(* PLC project LMM.project, Inovance company InoProShop(V1.9.1.6) InoProShop(V1.9.1.6) *)
(* stored: creationDateTime 2026-08-05T19:09:37.7446622, modificationDateTime 2026-08-05T19:09:08.6866302 *)

VAR_GLOBAL  (* GVL *)
  StartBtn AT %IX1.6 : BOOL;  (* 【面板启动】→ HMI_xStart *)
  StopBtn AT %IX1.4 : BOOL;  (* 【面板停止】→ HMI_xStop *)
  ResetBtn : BOOL;  (* 【面板复位】→ HMI_xStopHold3s；地址现场另绑 *)
  EStop AT %IX0.4 : BOOL;  (* 【面板急停】正常=TRUE 按下=FALSE *)
  StopLamp AT %QX0.6 : BOOL;  (* 【停止指示灯】← Dev_xStop *)
  StartLamp AT %QX0.7 : BOOL;  (* 【运行指示灯】← Dev_xRun *)
  JogFwd : BOOL;  (* 【面板前进】手动 X+ *)
  JogBwd : BOOL;  (* 【面板后退】手动 X- *)
  JogRight : BOOL;  (* 【面板右】手动 Y+ *)
  JogLeft : BOOL;  (* 【面板左】手动 Y- *)
  JogUp : BOOL;  (* 【面板上】手动 Z+ *)
  JogDown : BOOL;  (* 【面板下】手动 Z- *)
  JogClockAdd : BOOL;  (* 【面板顺时针】手动 R+ *)
  JogClockMis : BOOL;  (* 【面板逆时针】手动 R- *)
  HMI_xEStop : BOOL;  (* 【急停】TRUE正常 FALSE按下 = 物理 AND 触摸屏Req AND Web *)
  HMI_xStop : BOOL;  (* 【停止】任一源为真即停；长按3s=复位 *)
  HMI_xStopHold3s : BOOL;  (* 【复位】清急停锁存 + 轴故障复位 *)
  HMI_xStart : BOOL;  (* 【启动】上升沿 *)
  HMI_xEnable : BOOL;  (* 【启动别名】与 HMI_xStart 等效 *)
  xEStopLatched : BOOL;  (* 【急停锁存】仅复位可清 *)
  xFaultAggregate : BOOL;  (* 【故障汇总】任轴 ErrorStop *)
  eCtrlSrc : INT;  (* 【控制源】0=面板/触摸屏 1=远程Web；仅 PRG_TcpHmi 写 *)
  eOpMode : INT;  (* 【运行方式】0手动 1自动 *)
  iAlarmID : INT;  (* 【内部报警号】 *)
  HMI_eDevState : INT;  (* 【只读·状态码】0停 1运行 2错误 *)
  HMI_eOpMode : INT;  (* 【只读·方式显示】0手动 1自动 *)
  HMI_iAlarmShow : INT;  (* 【只读·报警号】1001急停 1002轴故障 1005力超时 1006从站失败 1007未就绪；1008已废 *)
  Dev_xStop : BOOL;  (* 【内部·停止派生】 *)
  Dev_xRun : BOOL;  (* 【内部·运行派生】 *)
  Dev_xError : BOOL;  (* 【内部·故障派生】 *)
  HMI_xDevStop : BOOL;  (* 【只读·停止灯】 *)
  HMI_xDevRun : BOOL;  (* 【只读·运行灯】 *)
  HMI_xDevError : BOOL;  (* 【只读·故障灯】 *)
  HMI_xLampEStop : BOOL;  (* 【只读·急停指示】 *)
  HMI_xLampEnableOk : BOOL;  (* 【只读·就绪灯】 *)
  HMI_xLampFault : BOOL;  (* 【只读·故障指示】 *)
  HMI_xAutoMode : BOOL;  (* 【模式】FALSE手动 TRUE自动 *)
  HMI_xJogXPos : BOOL;  (* 【X+】M1=M2 同速同向；与旋转互斥 *)
  HMI_xJogXNeg : BOOL;  (* 【X-】 *)
  HMI_xSpinLeft : BOOL;  (* 【左旋转】差速原地转；与 X± 互斥 *)
  HMI_xSpinRight : BOOL;  (* 【右旋转】 *)
  HMI_xJogYPos : BOOL;  (* 【Y+】受限位 *)
  HMI_xJogYNeg : BOOL;  (* 【Y-】 *)
  HMI_xJogZPos : BOOL;  (* 【Z+】回零后软限位 [-0.7,0] *)
  HMI_xJogZNeg : BOOL;  (* 【Z-】 *)
  HMI_xJogRPos : BOOL;  (* 【R+】需 xM5Ready *)
  HMI_xJogRNeg : BOOL;  (* 【R-】 *)
  HMI_xHomeY : BOOL;  (* 【Y回零】 *)
  HMI_xHomeZ : BOOL;  (* 【Z回零】完成后软限位生效 *)
  HMI_xHomeR : BOOL;  (* 【R回零】编码器回零 *)
  HMI_iHomeAxis : INT := 0;  (* 【回零轴选择】0无 1Y 2Z 3R *)
  HMI_xHomeExec : BOOL;  (* 【回零执行】对选定轴 *)
  HMI_xHomedY : BOOL;  (* 【只读·Y已回零】 *)
  HMI_xHomedZ : BOOL;  (* 【只读·Z已回零】 *)
  HMI_xHomedR : BOOL;  (* 【只读·R已回零】 *)
  HMI_xHomeBusyY : BOOL;  (* 【只读·Y回零中】 *)
  HMI_xHomeBusyZ : BOOL;  (* 【只读·Z回零中】 *)
  HMI_xHomeBusyR : BOOL;  (* 【只读·R回零中】 *)
  HMI_xAutoStart : BOOL;  (* 【自动启动】上升沿 *)
  HMI_xAutoAbort : BOOL;  (* 【自动中止】立即结束 *)
  HMI_rHeadingErr : REAL := 0.0;  (* 【航向误差】视觉/外部纠偏输入（实时量，不保持） *)
  iAutoStep : INT;  (* 【自动步】0Idle..6Done *)
  HMI_iAutoStepShow : INT;  (* 【只读·自动步号】 *)
  HMI_xAutoBusy : BOOL;  (* 【只读·自动忙】 *)
  HMI_xAutoDone : BOOL;  (* 【只读·自动完成】 *)
  Force_xEnable : BOOL := TRUE;  (* 【力通讯总使能】 *)
  Force_wInRaw AT %IW102 : WORD;  (* 组态读通道：0x0000 原始力 *)
  Force_wOutTare AT %QW42 : WORD;  (* 组态写通道：0x0011 去皮 *)
  Force_wOutUnit AT %QW43 : WORD := 5;  (* 组态写通道：0x0002 单位 5=N *)
  Force_rScale : REAL := 0.01;  (* 原始值倍率 *)
  Force_xReadTrig : BOOL;  (* 【内部·力读触发】组态用，勿绑屏 *)
  Force_xCommOk : BOOL;  (* 【只读·力通讯正常】 *)
  Force_xTimeout : BOOL;  (* 【只读·力超时】报警1005 *)
  Force_xSlaveFail : BOOL;  (* 【只读·从站使能失败】报警1006 *)
  Force_xTareBusy : BOOL;  (* 【只读·去皮中】 *)
  Force_xTareDone : BOOL;  (* 【只读·去皮完成】 *)
  Force_iRaw : INT;  (* 【只读·原始计数】 *)
  Force_iState : INT;  (* 【只读·力任务状态】 *)
  rForceAct : REAL;  (* 【实际力】N；Axis 任务写（模拟时 Logic 写） *)
  rForceKp : REAL;  (* 【内部·恒力Kp】 *)
  HMI_rForceSim : REAL;  (* 【力模拟值】N *)
  HMI_xForceSimEnable : BOOL;  (* 【力模拟使能】台架用 *)
  HMI_xForceTare : BOOL;  (* 【去皮】上升沿 *)
  HMI_xForceUntare : BOOL;  (* 【取消去皮】上升沿 *)
  HMI_xForceGuide : BOOL;  (* 【力引导电平】TRUE 持续 Z 恒力跟随 *)
  HMI_rForceShow : REAL;  (* 【只读·显示力】N *)
  Logic_xForceTare : BOOL;  (* 【内部·自动步去皮脉冲】 *)
  I_xLimYPos : BOOL;  (* 【Y正限位开关】 *)
  I_xLimYNeg : BOOL;  (* 【Y负限位开关】 *)
  I_xLimZPos : BOOL;  (* 【Z正限位开关】 *)
  I_xLimZNeg : BOOL;  (* 【Z负限位开关】 *)
  xIlk_BlockYPlus : BOOL;  (* 【联锁禁Y+】开关 ∨ Cfg 限位 *)
  xIlk_BlockYNeg : BOOL;  (* 【联锁禁Y-】 *)
  xIlk_BlockZPlus : BOOL;  (* 【联锁禁Z+】 *)
  xIlk_BlockZNeg : BOOL;  (* 【联锁禁Z-】 *)
  xM5Ready : BOOL := TRUE;  (* 【第5轴就绪】FALSE=忽略 R *)
  AxisCmd_xPower : BOOL;  (* 【轴使能】= 安全条件 *)
  AxisCmd_xStopAll : BOOL;  (* 【全停】急停/停止/故障/中止 *)
  AxisCmd_xResetFault : BOOL;  (* 【故障复位脉冲】 *)
  AxisCmd_xJogXPos : BOOL;  (* 【X+】 *)
  AxisCmd_xJogXNeg : BOOL;  (* 【X-】 *)
  AxisCmd_xSpinLeft : BOOL;  (* 【左旋】 *)
  AxisCmd_xSpinRight : BOOL;  (* 【右旋】 *)
  AxisCmd_xJogYPos : BOOL;  (* 【Y+】 *)
  AxisCmd_xJogYNeg : BOOL;  (* 【Y-】 *)
  AxisCmd_xJogZPos : BOOL;  (* 【Z+】 *)
  AxisCmd_xJogZNeg : BOOL;  (* 【Z-】 *)
  AxisCmd_xJogRPos : BOOL;  (* 【R+】 *)
  AxisCmd_xJogRNeg : BOOL;  (* 【R-】 *)
  AxisCmd_xHomeY : BOOL;  (* 【Y回零】完成/停止清 *)
  AxisCmd_xHomeZ : BOOL;  (* 【Z回零】 *)
  AxisCmd_xHomeR : BOOL;  (* 【R回零】 *)
  AxisCmd_xMoveRelX : BOOL;  (* 【X相对走距】速度模式+里程判完成 *)
  AxisCmd_rMoveDistX : REAL;  (* 【X相对距离】 *)
  AxisCmd_rMoveVelX : REAL;  (* 【X相对速度】 *)
  AxisCmd_xMoveRelY : BOOL;  (* 【Y相对】 *)
  AxisCmd_rMoveDistY : REAL;  (* 【Y相对距离】自动=跨距 *)
  AxisCmd_rMoveVelY : REAL;  (* 【Y速度】 *)
  AxisCmd_xMoveAbsY : BOOL;  (* 【Y绝对】归位用 *)
  AxisCmd_rMoveAbsPosY : REAL;  (* 【Y绝对目标】 *)
  AxisCmd_xForceFollow : BOOL;  (* 【Z力跟随】 *)
  AxisCmd_rForceSet : REAL;  (* 【力目标】 *)
  AxisCmd_rForceKp : REAL;  (* 【力Kp】 *)
  AxisCmd_rForceVelMax : REAL;  (* 【力跟随限速】 *)
  AxisCmd_xHoldR : BOOL;  (* 【R保持角】 *)
  AxisCmd_rRHoldPos : REAL;  (* 【R保持角位置】 *)
  AxisCmd_rHeadingErr : REAL;  (* 【航向误差】 *)
  AxisCmd_rTrackKp : REAL;  (* 【纠偏Kp】 *)
  AxisCmd_rJogVelX : REAL;  (* 【X点动速度】 *)
  AxisCmd_rSpinVel : REAL := 0.0;  (* 【旋转速度】 *)
  AxisCmd_rJogVelY : REAL;  (* 【Y点动速度】 *)
  AxisCmd_rJogVelZ : REAL;  (* 【Z点动速度】 *)
  AxisCmd_rJogVelR : REAL;  (* 【R点动速度】 *)
  AxisCmd_rWheelBase : REAL;  (* 【跨距】限幅 4..6 *)
  AxisCmd_rAccX : REAL;  (* 【X加速度】 *)
  AxisCmd_rDecX : REAL;  (* 【X减速度】 *)
  AxisCmd_rAccY : REAL;  (* 【Y加速度】 *)
  AxisCmd_rDecY : REAL;  (* 【Y减速度】 *)
  AxisCmd_rAccZ : REAL;  (* 【Z加速度】 *)
  AxisCmd_rDecZ : REAL;  (* 【Z减速度】 *)
  AxisCmd_rAccR : REAL;  (* 【R加速度】 *)
  AxisCmd_rDecR : REAL;  (* 【R减速度】 *)
  AxisFb_rVelCmdM1 : REAL;  (* 【只读·M1速度指令】含纠偏/旋转 *)
  AxisFb_rVelCmdM2 : REAL;  (* 【只读·M2速度指令】 *)
  AxisFb_rPosM1 : REAL;  (* 【只读·M1位置】 *)
  AxisFb_rPosM2 : REAL;  (* 【只读·M2位置】 *)
  AxisFb_rPosX : REAL;  (* 【只读·Virtual X 位置】走距判据 *)
  AxisFb_rSyncErr : REAL;  (* 【只读·M1-M2 同步误差】 *)
  AxisFb_rVelFactorX : REAL;  (* 【只读·Virtual Override 倍率】 *)
  AxisFb_xGantryCoupled : BOOL;  (* 【只读·龙门已 GearIn】M1且M2 *)
  AxisFb_xInGearM1 : BOOL;  (* 【只读·M1 电子齿轮 InGear】 *)
  AxisFb_xInGearM2 : BOOL;  (* 【只读·M2 电子齿轮 InGear】 *)
  AxisFb_xPoweredV : BOOL;  (* 【只读·Virtual 已使能】 *)
  AxisFb_xSyncWarn : BOOL;  (* 【只读·同步预警】 *)
  AxisFb_xSyncFault : BOOL;  (* 【只读·同步跳闸】已废，恒 FALSE *)
  AxisFb_iGantryState : INT;  (* 【只读·0Idle 1Coupling 2Coupled 3Decouple 4Diff 5Align】 *)
  AxisFb_rPosY : REAL;  (* 【只读·Y位置】 *)
  AxisFb_rPosZ : REAL;  (* 【只读·Z位置】 *)
  AxisFb_rPosR : REAL;  (* 【只读·R位置/角度】 *)
  AxisFb_xStandstill1 : BOOL;  (* 【只读·M1静止】 *)
  AxisFb_xStandstill2 : BOOL;  (* 【只读·M2静止】 *)
  AxisFb_xStandstillY : BOOL;  (* 【只读·Y静止】 *)
  AxisFb_xStandstillZ : BOOL;  (* 【只读·Z静止】 *)
  AxisFb_xStandstillR : BOOL;  (* 【只读·R静止】 *)
  AxisFb_xMovingM1 : BOOL;  (* 【只读·M1运动中】 *)
  AxisFb_xMovingM2 : BOOL;  (* 【只读·M2运动中】 *)
  AxisFb_xMovingY : BOOL;  (* 【只读·Y运动中】 *)
  AxisFb_xMovingZ : BOOL;  (* 【只读·Z运动中】 *)
  AxisFb_xMovingR : BOOL;  (* 【只读·R运动中】 *)
  AxisFb_xPoweredM1 : BOOL;  (* 【只读·M1已使能】 *)
  AxisFb_xPoweredM2 : BOOL;  (* 【只读·M2已使能】 *)
  AxisFb_xPoweredY : BOOL;  (* 【只读·Y已使能】 *)
  AxisFb_xPoweredZ : BOOL;  (* 【只读·Z已使能】 *)
  AxisFb_xPoweredR : BOOL;  (* 【只读·R已使能】 *)
  AxisFb_xReadyM1 : BOOL;  (* 【只读·M1就绪】 *)
  AxisFb_xReadyM2 : BOOL;  (* 【只读·M2就绪】 *)
  AxisFb_xReadyY : BOOL;  (* 【只读·Y就绪】 *)
  AxisFb_xReadyZ : BOOL;  (* 【只读·Z就绪】 *)
  AxisFb_xReadyR : BOOL;  (* 【只读·R就绪】 *)
  AxisFb_xReady : BOOL;  (* 【只读·全轴就绪】FALSE → 报警1007 *)
  AxisFb_xHomedY : BOOL;  (* 【只读·Y已回零】 *)
  AxisFb_xHomedZ : BOOL;  (* 【只读·Z已回零】 *)
  AxisFb_xHomedR : BOOL;  (* 【只读·R已回零】 *)
  AxisFb_xFaultM1 : BOOL;  (* 【只读·M1故障】 *)
  AxisFb_xFaultM2 : BOOL;  (* 【只读·M2故障】 *)
  AxisFb_xFaultY : BOOL;  (* 【只读·Y故障】 *)
  AxisFb_xFaultZ : BOOL;  (* 【只读·Z故障】 *)
  AxisFb_xFaultR : BOOL;  (* 【只读·R故障】 *)
  AxisFb_xMoveDoneX : BOOL;  (* 【只读·X走距完成】 *)
  AxisFb_xMoveDoneY : BOOL;  (* 【只读·Y完成】 *)
  MB_CmdIn AT %IW103 : ARRAY[0..63] OF WORD;  (* 【命令入】Holding 1000..1063 *)
  MB_StatusOut AT %QW44 : ARRAY[0..63] OF WORD;  (* 【状态出】Holding 1100..1163 *)
  Tcp_iCommStatus : INT;  (* 【只读·通讯诊断】0离线 1在线 2版本错 3序号错 4超时 *)
  Tcp_xConnected : BOOL;  (* 【只读·远程已连接】 *)
  Tcp_xTimeout : BOOL;  (* 【只读·远程超时】 *)
  Tcp_xOnline : BOOL;  (* 【只读·远程在线可用】 *)
  Tcp_wLastHb : WORD;  (* 【内部·上次心跳】 *)
  Tcp_wLastSeq : WORD;  (* 【内部·上次命令序号】 *)
  Tcp_wStatusSeq : WORD;  (* 【内部·状态序号】 *)
  Tcp_xEStop : BOOL := TRUE;  (* 【Web影子·急停】掉线强制 TRUE *)
  Tcp_xStop : BOOL;  (* 【Web影子·停止】 *)
  Tcp_xStopHold3s : BOOL;  (* 【Web影子·复位】 *)
  Tcp_xStart : BOOL;  (* 【Web影子·启动】 *)
  Tcp_xEnable : BOOL;  (* 【Web影子·启动别名】 *)
  Tcp_xAutoMode : BOOL;  (* 【Web影子·模式】 *)
  Tcp_xJogXPos : BOOL;  (* 【Web影子·X+】 *)
  Tcp_xJogXNeg : BOOL;  (* 【Web影子·X-】 *)
  Tcp_xSpinLeft : BOOL;  (* 【Web影子·左旋】 *)
  Tcp_xSpinRight : BOOL;  (* 【Web影子·右旋】 *)
  Tcp_xJogYPos : BOOL;  (* 【Web影子·Y+】 *)
  Tcp_xJogYNeg : BOOL;  (* 【Web影子·Y-】 *)
  Tcp_xJogZPos : BOOL;  (* 【Web影子·Z+】 *)
  Tcp_xJogZNeg : BOOL;  (* 【Web影子·Z-】 *)
  Tcp_xJogRPos : BOOL;  (* 【Web影子·R+】 *)
  Tcp_xJogRNeg : BOOL;  (* 【Web影子·R-】 *)
  Tcp_xHomeY : BOOL;  (* 【Web影子·Y回零】 *)
  Tcp_xHomeZ : BOOL;  (* 【Web影子·Z回零】 *)
  Tcp_xHomeR : BOOL;  (* 【Web影子·R回零】 *)
  Tcp_iHomeAxis : INT := 0;  (* 【Web影子·回零轴选择】 *)
  Tcp_xHomeExec : BOOL;  (* 【Web影子·回零执行】 *)
  Tcp_rJogVelX : REAL := 0.4;  (* 【Web影子·X速度】 *)
  Tcp_rSpinVel : REAL := 0.3;  (* 【Web影子·旋转速度】 *)
  Tcp_rJogVelY : REAL := 0.3;  (* 【Web影子·Y速度】 *)
  Tcp_rJogVelZ : REAL := 0.2;  (* 【Web影子·Z速度】 *)
  Tcp_rJogVelR : REAL := 0.2;  (* 【Web影子·R速度】 *)
  Tcp_xAutoStart : BOOL;  (* 【Web影子·自动启动】 *)
  Tcp_xAutoAbort : BOOL;  (* 【Web影子·自动中止】 *)
  Tcp_rAutoDistX : REAL := 1.0;  (* 【Web影子·自动X距】 *)
  Tcp_rAutoVelX : REAL := 0.4;  (* 【Web影子·自动X速】 *)
  Tcp_rAutoVelY : REAL := 0.3;  (* 【Web影子·自动Y速】 *)
  Tcp_rAutoVelZ : REAL := 0.15;  (* 【Web影子·自动Z速】 *)
  Tcp_rWheelBase : REAL := 5.0;  (* 【Web影子·跨距】 *)
  Tcp_rForceSet : REAL := 100.0;  (* 【Web影子·力设定】 *)
  Tcp_xForceSimEnable : BOOL := FALSE;  (* 【Web影子·力模拟使能】 *)
  Tcp_rForceSim : REAL;  (* 【Web影子·力模拟值】 *)
  Tcp_xForceTare : BOOL;  (* 【Web影子·去皮】 *)
  Tcp_xForceUntare : BOOL;  (* 【Web影子·取消去皮】 *)
  Tcp_xForceGuide : BOOL;  (* 【Web影子·力引导】 *)
  Tcp_iAutoPasses : INT := 1;  (* 【Web影子·自动道数】 *)
  Tcp_rHeadingErr : REAL := 0.0;  (* 【Web影子·航向误差】 *)
  Tcp_rKpTrack : REAL;  (* 【Web影子·纠偏Kp】 *)
  Tcp_rKpForce : REAL;  (* 【Web影子·力Kp】 *)
  Tcp_rAccX : REAL := 100.0;  (* 【Web影子·X加速度】 *)
  Tcp_rDecX : REAL := 100.0;  (* 【Web影子·X减速度】 *)
  Tcp_rAccY : REAL := 100.0;  (* 【Web影子·Y加速度】 *)
  Tcp_rDecY : REAL := 100.0;  (* 【Web影子·Y减速度】 *)
  Tcp_rAccZ : REAL := 100.0;  (* 【Web影子·Z加速度】 *)
  Tcp_rDecZ : REAL := 100.0;  (* 【Web影子·Z减速度】 *)
  Tcp_rAccR : REAL := 100.0;  (* 【Web影子·R加速度】 *)
  Tcp_rDecR : REAL := 100.0;  (* 【Web影子·R减速度】 *)
  HMI_xStartReq : BOOL;  (* 【触摸屏启动】 *)
  HMI_xStopReq : BOOL;  (* 【触摸屏停止】 *)
  HMI_xResetReq : BOOL;  (* 【触摸屏复位】 *)
  HMI_xEStopReq : BOOL := TRUE;  (* 【触摸屏急停】TRUE正常 *)
  HMI_xAutoStartReq : BOOL;  (* 【触摸屏自动启动】 *)
  HMI_xAutoAbortReq : BOOL;  (* 【触摸屏自动中止】 *)
  {attribute 'retain'}
  HMI_rJogVelX : REAL := 0.4;  (* 【X直行速度】与旋转速度分开 *)
  {attribute 'retain'}
  HMI_rSpinVel : REAL := 0.3;  (* 【左右旋速度】 *)
  {attribute 'retain'}
  HMI_rJogVelY : REAL := 0.4;  (* 【Y点动速度】 *)
  {attribute 'retain'}
  HMI_rJogVelZ : REAL := 0.4;  (* 【Z点动速度】力跟随限速后备 *)
  {attribute 'retain'}
  HMI_rJogVelR : REAL := 0.2;  (* 【R点动速度】 *)
  {attribute 'retain'}
  HMI_rAccX : REAL := 25;  (* 【X加速度】 *)
  {attribute 'retain'}
  HMI_rDecX : REAL := 25;  (* 【X减速度】 *)
  {attribute 'retain'}
  HMI_rAccY : REAL := 25;  (* 【Y加速度】 *)
  {attribute 'retain'}
  HMI_rDecY : REAL := 25;  (* 【Y减速度】 *)
  {attribute 'retain'}
  HMI_rAccZ : REAL := 25;  (* 【Z加速度】 *)
  {attribute 'retain'}
  HMI_rDecZ : REAL := 25;  (* 【Z减速度】 *)
  {attribute 'retain'}
  HMI_rAccR : REAL := 25;  (* 【R加速度】 *)
  {attribute 'retain'}
  HMI_rDecR : REAL := 25;  (* 【R减速度】 *)
  {attribute 'retain'}
  HMI_rAutoDistX : REAL := 1.0;  (* 【自动X走距】每道 *)
  {attribute 'retain'}
  HMI_rAutoVelX : REAL := 0.4;  (* 【自动X速度】 *)
  {attribute 'retain'}
  HMI_rAutoVelY : REAL := 0.3;  (* 【自动Y速度】 *)
  {attribute 'retain'}
  HMI_rAutoVelZ : REAL := 0.15;  (* 【自动Z速度】力跟随限速参考 *)
  {attribute 'retain'}
  HMI_rWheelBase : REAL := 5.0;  (* 【龙门跨距=Y行程】4~6 m *)
  {attribute 'retain'}
  HMI_iAutoPasses : INT := 1;  (* 【自动总道数】≥1 *)
  {attribute 'retain'}
  HMI_rForceSet : REAL := 100.0;  (* 【恒力设定】N *)
  {attribute 'retain'}
  HMI_rKpForce : REAL := 1.0;  (* 【力跟随Kp】 *)
  {attribute 'retain'}
  HMI_rKpTrack : REAL := 0.0;  (* 【直线纠偏Kp】 *)
  {attribute 'retain'}
  Cfg_rLimYPos : REAL := 6.0;  (* 【Y正限位】m，默认跨距上限 *)
  {attribute 'retain'}
  Cfg_rLimYNeg : REAL := 0.0;  (* 【Y负限位】m *)
  {attribute 'retain'}
  Cfg_rLimZPos : REAL := 0.0;  (* 【Z正限位】上 *)
  {attribute 'retain'}
  Cfg_rLimZNeg : REAL := -0.7;  (* 【Z负限位】下压行程 *)
  {attribute 'retain'}
  Cfg_rLimRPos : REAL := 180.0;  (* 【R正限位】度 *)
  {attribute 'retain'}
  Cfg_rLimRNeg : REAL := -180.0;  (* 【R负限位】度 *)
  {attribute 'retain'}
  Cfg_rVelBaseMaxX : REAL := 1.0;  (* 【X速度基准】诊断倍率分母；≥最大 Jog/Auto *)
  {attribute 'retain'}
  Cfg_rPhaseMax : REAL := 0.01;  (* 【跟轨相位限幅】u；连续 Phasing *)
  {attribute 'retain'}
  Cfg_rSyncWarn : REAL := 0.02;  (* 【同步预警】|M1-M2|；降速 *)
  {attribute 'retain'}
  Cfg_rSyncFault : REAL := 0.05;  (* 【同步跳闸】已废；保留 RETAIN 布局 *)
END_VAR

PROGRAM PRG_Logic
  VAR
    tonHold : TON;
    tonReady : TON;
    xResetPulse : BOOL;
    xResetPrev : BOOL;
    xSafe : BOOL;
    xAutoStartPrev : BOOL;
    xAutoStartEdge : BOOL;
    rRHold : REAL;
    iPass : INT;
    xAutoTareSent : BOOL;
    xHomeTrigY : BOOL;
    xHomeTrigZ : BOOL;
    xHomeTrigR : BOOL;
    xHomeTrigYPrev : BOOL;
    xHomeTrigZPrev : BOOL;
    xHomeTrigRPrev : BOOL;
    xAnyHomeBusy : BOOL;
    xReadyAll : BOOL;
    xPanelSrc : BOOL;  (* eCtrlSrc=0：面板/触摸屏源 *)
    xJogXPosM : BOOL;  (* 合并后点动（HMI/Web OR 面板键） *)
    xJogXNegM : BOOL;
    xJogYPosM : BOOL;
    xJogYNegM : BOOL;
    xJogZPosM : BOOL;
    xJogZNegM : BOOL;
    xJogRPosM : BOOL;
    xJogRNegM : BOOL;
  END_VAR

            (* PRG_Logic — 消费已仲裁 HMI_* + 面板键；写 AxisCmd_*；状态只读派生（无状态机耦合）。
   禁止 CALL Axis / FB_Servo。 *)

(* ===== 急停锁存 / 长按复位 ===== *)
IF NOT HMI_xEStop THEN
    xEStopLatched := TRUE;
END_IF;
tonHold(IN := HMI_xStop AND HMI_xEStop, PT := T#3S);
xResetPulse := (HMI_xStopHold3s OR tonHold.Q) AND NOT xResetPrev;
xResetPrev := HMI_xStopHold3s OR tonHold.Q;
IF xResetPulse THEN
    xEStopLatched := FALSE;
    AxisCmd_xResetFault := TRUE;
    iAutoStep := 0;
    iPass := 0;
    Force_xSlaveFail := FALSE;
ELSE
    AxisCmd_xResetFault := FALSE;
END_IF;

(* 故障汇总：各轴 Errorstop（同步跳闸已废，不再 OR AxisFb_xSyncFault） *)
xFaultAggregate := AxisFb_xFaultM1 OR AxisFb_xFaultM2 OR AxisFb_xFaultY OR AxisFb_xFaultZ
    OR (xM5Ready AND AxisFb_xFaultR);

IF HMI_xAutoMode THEN eOpMode := 1; ELSE eOpMode := 0; END_IF;
HMI_eOpMode := eOpMode;

(* 安全 / 使能 —— 去耦：只看急停 + 故障 *)
xSafe := HMI_xEStop AND NOT xEStopLatched;
AxisCmd_xPower := xSafe;
AxisCmd_xStopAll := HMI_xStop OR NOT xSafe OR xFaultAggregate OR HMI_xAutoAbort;

(* 力/纠偏参数下发 *)
rForceKp := HMI_rKpForce;
IF rForceKp < 1.0E-6 THEN rForceKp := 1.0; END_IF;
AxisCmd_rForceSet := HMI_rForceSet;
AxisCmd_rForceKp := rForceKp;
AxisCmd_rForceVelMax := ABS(HMI_rAutoVelZ);
IF AxisCmd_rForceVelMax < 1.0E-6 THEN AxisCmd_rForceVelMax := ABS(HMI_rJogVelZ); END_IF;
AxisCmd_rHeadingErr := HMI_rHeadingErr;

IF HMI_xForceSimEnable THEN
    rForceAct := HMI_rForceSim;
END_IF;
HMI_rForceShow := rForceAct;

AxisCmd_rJogVelX := HMI_rJogVelX;
AxisCmd_rSpinVel := HMI_rSpinVel;
AxisCmd_rJogVelY := HMI_rJogVelY;
AxisCmd_rJogVelZ := HMI_rJogVelZ;
AxisCmd_rJogVelR := HMI_rJogVelR;
AxisCmd_rWheelBase := LIMIT(4.0, HMI_rWheelBase, 6.0);
(* 每轴加减速（RETAIN 参数；<1 时兜底 100） *)
AxisCmd_rAccX := HMI_rAccX; IF AxisCmd_rAccX < 1.0 THEN AxisCmd_rAccX := 100.0; END_IF;
AxisCmd_rDecX := HMI_rDecX; IF AxisCmd_rDecX < 1.0 THEN AxisCmd_rDecX := 100.0; END_IF;
AxisCmd_rAccY := HMI_rAccY; IF AxisCmd_rAccY < 1.0 THEN AxisCmd_rAccY := 100.0; END_IF;
AxisCmd_rDecY := HMI_rDecY; IF AxisCmd_rDecY < 1.0 THEN AxisCmd_rDecY := 100.0; END_IF;
AxisCmd_rAccZ := HMI_rAccZ; IF AxisCmd_rAccZ < 1.0 THEN AxisCmd_rAccZ := 100.0; END_IF;
AxisCmd_rDecZ := HMI_rDecZ; IF AxisCmd_rDecZ < 1.0 THEN AxisCmd_rDecZ := 100.0; END_IF;
AxisCmd_rAccR := HMI_rAccR; IF AxisCmd_rAccR < 1.0 THEN AxisCmd_rAccR := 100.0; END_IF;
AxisCmd_rDecR := HMI_rDecR; IF AxisCmd_rDecR < 1.0 THEN AxisCmd_rDecR := 100.0; END_IF;

(* 限位联锁：物理限位输入 ∨ 可配置硬限位（Cfg_rLim*，FB_Servo 内另有最终闸门） *)
xIlk_BlockYPlus := I_xLimYPos OR (AxisFb_rPosY >= Cfg_rLimYPos);
xIlk_BlockYNeg := I_xLimYNeg OR (AxisFb_rPosY <= Cfg_rLimYNeg);
xIlk_BlockZPlus := I_xLimZPos OR (AxisFb_rPosZ >= Cfg_rLimZPos);
xIlk_BlockZNeg := I_xLimZNeg OR (AxisFb_rPosZ <= Cfg_rLimZNeg);

(* 每拍清命令 *)
AxisCmd_xJogXPos := FALSE; AxisCmd_xJogXNeg := FALSE;
AxisCmd_xSpinLeft := FALSE; AxisCmd_xSpinRight := FALSE;
AxisCmd_xJogYPos := FALSE; AxisCmd_xJogYNeg := FALSE;
AxisCmd_xJogZPos := FALSE; AxisCmd_xJogZNeg := FALSE;
AxisCmd_xJogRPos := FALSE; AxisCmd_xJogRNeg := FALSE;
AxisCmd_xForceFollow := FALSE;
AxisCmd_xMoveRelX := FALSE;
AxisCmd_xMoveRelY := FALSE;
AxisCmd_xMoveAbsY := FALSE;
AxisCmd_xHoldR := FALSE;
AxisCmd_rTrackKp := 0.0;
Logic_xForceTare := FALSE;

xAutoStartEdge := HMI_xAutoStart AND NOT xAutoStartPrev;
xAutoStartPrev := HMI_xAutoStart;

IF HMI_xAutoAbort OR NOT xSafe OR xFaultAggregate THEN
    iAutoStep := 0;
    iPass := 0;
    HMI_xAutoBusy := FALSE;
END_IF;

(* ===== 点动源合并：面板键（仅面板/触摸屏源时）OR 触摸屏/Web ===== *)
xPanelSrc := (eCtrlSrc = 0);
xJogXPosM := HMI_xJogXPos OR (xPanelSrc AND JogFwd);
xJogXNegM := HMI_xJogXNeg OR (xPanelSrc AND JogBwd);
xJogYPosM := HMI_xJogYPos OR (xPanelSrc AND JogRight);
xJogYNegM := HMI_xJogYNeg OR (xPanelSrc AND JogLeft);
xJogZPosM := HMI_xJogZPos OR (xPanelSrc AND JogUp);
xJogZNegM := HMI_xJogZNeg OR (xPanelSrc AND JogDown);
xJogRPosM := HMI_xJogRPos OR (xPanelSrc AND JogClockAdd);
xJogRNegM := HMI_xJogRNeg OR (xPanelSrc AND JogClockMis);

(* ===== 手动 ===== *)
IF xSafe AND (eOpMode = 0) AND NOT HMI_xStop AND NOT xFaultAggregate THEN
    IF HMI_xSpinLeft XOR HMI_xSpinRight THEN
        AxisCmd_xSpinLeft := HMI_xSpinLeft;
        AxisCmd_xSpinRight := HMI_xSpinRight;
    ELSIF xJogXPosM XOR xJogXNegM THEN
        AxisCmd_xJogXPos := xJogXPosM;
        AxisCmd_xJogXNeg := xJogXNegM;
    END_IF;
    AxisCmd_xJogYPos := xJogYPosM AND NOT xIlk_BlockYPlus;
    AxisCmd_xJogYNeg := xJogYNegM AND NOT xIlk_BlockYNeg;
    IF HMI_xForceGuide THEN
        AxisCmd_xForceFollow := TRUE;
    ELSE
        AxisCmd_xJogZPos := xJogZPosM AND NOT xIlk_BlockZPlus;
        AxisCmd_xJogZNeg := xJogZNegM AND NOT xIlk_BlockZNeg;
    END_IF;
    IF xM5Ready THEN
        AxisCmd_xJogRPos := xJogRPosM;
        AxisCmd_xJogRNeg := xJogRNegM;
    END_IF;
END_IF;

(* ===== 自动多道循环 ===== *)
IF xSafe AND (eOpMode = 1) AND NOT HMI_xStop AND NOT xFaultAggregate THEN
    IF iAutoStep = 0 AND xAutoStartEdge THEN
        rRHold := AxisFb_rPosR;
        xAutoTareSent := FALSE;
        HMI_xAutoDone := FALSE;
        HMI_xAutoBusy := TRUE;
        iPass := 1;
        iAutoStep := 1;
    END_IF;

    CASE iAutoStep OF
        1:
            AxisCmd_xHoldR := TRUE;
            AxisCmd_rRHoldPos := rRHold;
            AxisCmd_rTrackKp := HMI_rKpTrack;
            AxisCmd_rMoveDistX := HMI_rAutoDistX;
            AxisCmd_rMoveVelX := HMI_rAutoVelX;
            AxisCmd_xMoveRelX := TRUE;
            IF AxisFb_xMoveDoneX THEN
                AxisCmd_xMoveRelX := FALSE;
                iAutoStep := 2;
            END_IF;
        2:
            AxisCmd_xHoldR := TRUE;
            AxisCmd_rRHoldPos := rRHold;
            AxisCmd_rMoveAbsPosY := 0.0;
            AxisCmd_rMoveVelY := HMI_rAutoVelY;
            AxisCmd_xMoveAbsY := TRUE;
            IF AxisFb_xStandstillY AND (ABS(AxisFb_rPosY) < 0.005) THEN
                AxisCmd_xMoveAbsY := FALSE;
                xAutoTareSent := FALSE;
                iAutoStep := 3;
            END_IF;
        3:
            AxisCmd_xHoldR := TRUE;
            AxisCmd_rRHoldPos := rRHold;
            IF NOT xAutoTareSent THEN
                Logic_xForceTare := TRUE;
                xAutoTareSent := TRUE;
            END_IF;
            AxisCmd_xForceFollow := TRUE;
            IF rForceAct >= HMI_rForceSet THEN
                iAutoStep := 4;
            END_IF;
        4:
            AxisCmd_xHoldR := TRUE;
            AxisCmd_rRHoldPos := rRHold;
            AxisCmd_xForceFollow := TRUE;
            AxisCmd_rMoveDistY := AxisCmd_rWheelBase;
            AxisCmd_rMoveVelY := HMI_rAutoVelY;
            AxisCmd_xMoveRelY := TRUE;
            IF AxisFb_xMoveDoneY THEN
                AxisCmd_xMoveRelY := FALSE;
                iAutoStep := 5;
            END_IF;
        5:
            IF iPass < HMI_iAutoPasses THEN
                iPass := iPass + 1;
                iAutoStep := 1;
            ELSE
                iAutoStep := 6;
            END_IF;
        6:
            HMI_xAutoBusy := FALSE;
            HMI_xAutoDone := TRUE;
            iAutoStep := 0;
            iPass := 0;
    END_CASE;
END_IF;

(* ===== 回零：Y/Z/R；同时只回一轴 ===== *)
xHomeTrigY := HMI_xHomeY OR ((HMI_iHomeAxis = 1) AND HMI_xHomeExec);
xHomeTrigZ := HMI_xHomeZ OR ((HMI_iHomeAxis = 2) AND HMI_xHomeExec);
xHomeTrigR := HMI_xHomeR OR ((HMI_iHomeAxis = 3) AND HMI_xHomeExec);
xAnyHomeBusy := AxisCmd_xHomeY OR AxisCmd_xHomeZ OR AxisCmd_xHomeR;

IF AxisCmd_xStopAll OR NOT xSafe OR xFaultAggregate THEN
    AxisCmd_xHomeY := FALSE;
    AxisCmd_xHomeZ := FALSE;
    AxisCmd_xHomeR := FALSE;
ELSE
    IF AxisCmd_xHomeY AND AxisFb_xHomedY THEN AxisCmd_xHomeY := FALSE; END_IF;
    IF AxisCmd_xHomeZ AND AxisFb_xHomedZ THEN AxisCmd_xHomeZ := FALSE; END_IF;
    IF AxisCmd_xHomeR AND AxisFb_xHomedR THEN AxisCmd_xHomeR := FALSE; END_IF;
    IF (eOpMode = 0) AND NOT HMI_xStop THEN
        IF xHomeTrigY AND NOT xHomeTrigYPrev AND NOT xAnyHomeBusy THEN
            AxisCmd_xHomeY := TRUE;
        ELSIF xHomeTrigZ AND NOT xHomeTrigZPrev AND NOT xAnyHomeBusy THEN
            AxisCmd_xHomeZ := TRUE;
        ELSIF xHomeTrigR AND NOT xHomeTrigRPrev AND NOT xAnyHomeBusy AND xM5Ready THEN
            AxisCmd_xHomeR := TRUE;
        END_IF;
    END_IF;
END_IF;
xHomeTrigYPrev := xHomeTrigY;
xHomeTrigZPrev := xHomeTrigZ;
xHomeTrigRPrev := xHomeTrigR;

IF AxisCmd_xHomeY THEN AxisCmd_xJogYPos := FALSE; AxisCmd_xJogYNeg := FALSE; END_IF;
IF AxisCmd_xHomeZ THEN AxisCmd_xJogZPos := FALSE; AxisCmd_xJogZNeg := FALSE; AxisCmd_xForceFollow := FALSE; END_IF;
IF AxisCmd_xHomeR THEN AxisCmd_xJogRPos := FALSE; AxisCmd_xJogRNeg := FALSE; END_IF;

HMI_xHomedY := AxisFb_xHomedY;
HMI_xHomedZ := AxisFb_xHomedZ;
HMI_xHomedR := AxisFb_xHomedR;
HMI_xHomeBusyY := AxisCmd_xHomeY;
HMI_xHomeBusyZ := AxisCmd_xHomeZ;
HMI_xHomeBusyR := AxisCmd_xHomeR;

(* 使能就绪诊断 → 1007 *)
xReadyAll := AxisFb_xReadyM1 AND AxisFb_xReadyM2 AND AxisFb_xReadyY AND AxisFb_xReadyZ
    AND (NOT xM5Ready OR AxisFb_xReadyR);
tonReady(IN := AxisCmd_xPower AND NOT xReadyAll AND NOT xFaultAggregate, PT := T#2S);

(* 报警 *)
IF xEStopLatched OR NOT HMI_xEStop THEN
    iAlarmID := 1001;
ELSIF AxisFb_xFaultM1 OR AxisFb_xFaultM2 OR AxisFb_xFaultY OR AxisFb_xFaultZ
        OR (xM5Ready AND AxisFb_xFaultR) THEN
    iAlarmID := 1002;
ELSIF tonReady.Q THEN
    iAlarmID := 1007;
ELSIF NOT HMI_xForceSimEnable AND Force_xSlaveFail THEN
    iAlarmID := 1006;
ELSIF NOT HMI_xForceSimEnable AND Force_xTimeout THEN
    iAlarmID := 1005;
ELSE
    iAlarmID := 0;
END_IF;

(* 状态灯（只读派生，不互锁） *)
Dev_xError := xFaultAggregate;
Dev_xRun := xSafe AND NOT HMI_xStop AND NOT xFaultAggregate;
Dev_xStop := NOT Dev_xRun AND NOT Dev_xError;
HMI_xDevError := Dev_xError;
HMI_xDevRun := Dev_xRun;
HMI_xDevStop := Dev_xStop;
IF Dev_xError THEN HMI_eDevState := 2;
ELSIF Dev_xRun THEN HMI_eDevState := 1;
ELSE HMI_eDevState := 0; END_IF;

HMI_iAutoStepShow := iAutoStep;
HMI_xLampEStop := xEStopLatched OR NOT HMI_xEStop;
HMI_xLampEnableOk := Dev_xRun;
HMI_xLampFault := xFaultAggregate;
HMI_iAlarmShow := iAlarmID;

StopLamp := Dev_xStop;
StartLamp := Dev_xRun;
          
END_PROGRAM

PROGRAM PRG_Force485
  VAR
    iSlaveStep : INT;
    iSlaveTry : INT;
    tonSlave : TON;
    wSnap : WORD;
    wRawLast : WORD;
    xTarePrev : BOOL;
    xUntarePrev : BOOL;
    xUnitInit : BOOL;
    diRaw : DINT;
    rTmp : REAL;
    xTareReq : BOOL;
  END_VAR

            (*==============================================================================
 * PRG_Force485 — SM1001 使能 + 发读等回文（最多3次）+ 去皮/换算
 *
 * 流程（严格按需求）：
 *   1) 使能 Modbus 从站 SM1001
 *   2) 发送一次读（破坏 Force_wInRaw 快照，等组态 FC03 通道写回 = 有回文）
 *   3) 有回文 → Force_xCommOk，进入成功态，不再重试
 *   4) 无回文 → 关闭 SM1001，重新使能，再读
 *   5) 3 次均无回文 → Force_xSlaveFail / 报警 1006
 *
 * 组态：读通道 FC03 0x0000 → Force_wInRaw（循环或由 Force_xReadTrig 触发均可）
 *============================================================================*)

Force_xTareDone := FALSE;

IF NOT Force_xEnable THEN
	SM1001 := FALSE;
	Force_xReadTrig := FALSE;
	Force_xCommOk := FALSE;
	Force_xTimeout := FALSE;
	Force_xTareBusy := FALSE;
	Force_xSlaveFail := FALSE;
	Force_iState := 0;
	iSlaveStep := 0;
	iSlaveTry := 0;
	RETURN;
END_IF;

CASE iSlaveStep OF
	0: (* 准备：先关从站，再进入使能 *)
		IF iSlaveTry >= 3 THEN
			SM1001 := FALSE;
			Force_xReadTrig := FALSE;
			Force_xSlaveFail := TRUE;
			Force_xTimeout := TRUE;
			Force_xCommOk := FALSE;
			Force_iState := -2;
			iSlaveStep := 99;
		ELSE
			SM1001 := FALSE;
			Force_xReadTrig := FALSE;
			Force_xCommOk := FALSE;
			tonSlave(IN := FALSE);
			tonSlave(IN := TRUE, PT := T#200MS);
			Force_iState := 0;
			iSlaveStep := 1;
		END_IF;

	1: (* 关断保持 *)
		SM1001 := FALSE;
		Force_xReadTrig := FALSE;
		tonSlave();
		IF tonSlave.Q THEN
			tonSlave(IN := FALSE);
			iSlaveStep := 2;
		END_IF;

	2: (* ① 使能从站 *)
		SM1001 := TRUE;
		Force_xReadTrig := FALSE;
		iSlaveTry := iSlaveTry + 1;
		tonSlave(IN := FALSE);
		tonSlave(IN := TRUE, PT := T#100MS);
		Force_iState := 1;
		iSlaveStep := 3;

	3: (* 使能稳定后：② 发读命令（破坏快照 + 读触发） *)
		SM1001 := TRUE;
		tonSlave();
		IF tonSlave.Q THEN
			(* 破坏映射值：有回文时通道会写回真实寄存器 *)
			wSnap := Force_wInRaw XOR 16#FFFF;
			Force_wInRaw := wSnap;
			Force_xReadTrig := FALSE;
			tonSlave(IN := FALSE);
			tonSlave(IN := TRUE, PT := T#20MS);
			Force_iState := 2;
			iSlaveStep := 4;
		END_IF;

	4: (* 读触发上升沿 *)
		SM1001 := TRUE;
		tonSlave();
		IF tonSlave.Q THEN
			Force_xReadTrig := TRUE;
			tonSlave(IN := FALSE);
			tonSlave(IN := TRUE, PT := T#500MS);
			Force_iState := 3;
			iSlaveStep := 5;
		END_IF;

	5: (* ③ 等回文：Force_wInRaw 被总线写回且不等于破坏值 *)
		SM1001 := TRUE;
		Force_xReadTrig := TRUE;
		tonSlave();
		IF Force_wInRaw <> wSnap THEN
			(* 有回文 → 成功，不再尝试 *)
			Force_xReadTrig := FALSE;
			Force_xCommOk := TRUE;
			Force_xTimeout := FALSE;
			Force_xSlaveFail := FALSE;
			wRawLast := Force_wInRaw;
			Force_iState := 4;
			tonSlave(IN := FALSE);
			iSlaveStep := 10;
		ELSIF tonSlave.Q THEN
			(* 无回文 → 关从站，回到 0 重新使能 *)
			Force_xReadTrig := FALSE;
			SM1001 := FALSE;
			Force_xCommOk := FALSE;
			Force_iState := 5;
			tonSlave(IN := FALSE);
			iSlaveStep := 0;
		END_IF;

	10: (* 成功：保持使能，不再重试使能 *)
		SM1001 := TRUE;
		Force_xReadTrig := FALSE;
		Force_xCommOk := TRUE;
		Force_xTimeout := FALSE;
		IF Force_wInRaw <> wRawLast THEN
			wRawLast := Force_wInRaw;
		END_IF;

	99: (* 3 次失败；复位清 Force_xSlaveFail 后从 0 重来 *)
		SM1001 := FALSE;
		Force_xReadTrig := FALSE;
		IF Force_xSlaveFail THEN
			Force_xTimeout := TRUE;
			Force_xCommOk := FALSE;
		ELSE
			iSlaveTry := 0;
			Force_xTimeout := FALSE;
			iSlaveStep := 0;
		END_IF;
END_CASE;

(* ----- 原始值换算（成功后持续；探测中也换算便于监视） ----- *)
diRaw := DWORD_TO_DINT(WORD_TO_DWORD(Force_wInRaw));
IF diRaw > 32767 THEN
	diRaw := diRaw - 65536;
END_IF;
Force_iRaw := DINT_TO_INT(diRaw);
IF Force_rScale < 1.0E-12 THEN
	rTmp := INT_TO_REAL(Force_iRaw);
ELSE
	rTmp := INT_TO_REAL(Force_iRaw) * Force_rScale;
END_IF;
IF NOT HMI_xForceSimEnable AND iSlaveStep = 10 THEN
	rForceAct := rTmp;
END_IF;

IF NOT xUnitInit AND iSlaveStep = 10 THEN
	Force_wOutUnit := 5;
	xUnitInit := TRUE;
END_IF;

xTareReq := FALSE;
IF iSlaveStep = 10 THEN
	IF ((HMI_xForceTare OR Tcp_xForceTare OR Logic_xForceTare) AND NOT xTarePrev) THEN
		Force_wOutTare := 1;
		xTareReq := TRUE;
		Force_xTareDone := TRUE;
	END_IF;
	xTarePrev := HMI_xForceTare OR Tcp_xForceTare OR Logic_xForceTare;
	IF Tcp_xForceTare THEN
		Tcp_xForceTare := FALSE;
	END_IF;
	IF Logic_xForceTare THEN
		Logic_xForceTare := FALSE;
	END_IF;

	IF ((HMI_xForceUntare OR Tcp_xForceUntare) AND NOT xUntarePrev) THEN
		Force_wOutTare := 2;
		xTareReq := TRUE;
		Force_xTareDone := TRUE;
	END_IF;
	xUntarePrev := HMI_xForceUntare OR Tcp_xForceUntare;
	IF Tcp_xForceUntare THEN
		Tcp_xForceUntare := FALSE;
	END_IF;
END_IF;

Force_xTareBusy := xTareReq;

          
END_PROGRAM

PROGRAM PLC_PRG

            (* MainTask 入口：HMI 交互 -> 设备逻辑；PRG_Axis_Control 在 ETHERCAT 任务独立运行 *)
PRG_TcpHmi();
PRG_Logic();
PRG_Force485();
          
END_PROGRAM

FUNCTION_BLOCK FB_XLineTrack
  VAR_INPUT
    xEnable : BOOL;
    xStop : BOOL;
    eMode : INT;
    rBaseVel : REAL;  (* 直行基础速度（可正可负） *)
    rSpinVel : REAL;  (* 原地旋转速度（正值） *)
    rHeadingErr : REAL;  (* 航向误差（视觉/外部；手动传 0） *)
    rKpTrack : REAL;  (* 纠偏 Kp *)
    rTrimMax : REAL;  (* 纠偏限幅 *)
  END_VAR
  VAR_OUTPUT
    rVelM1 : REAL;  (* M1 速度指令 *)
    rVelM2 : REAL;  (* M2 速度指令 *)
    xActive : BOOL;
  END_VAR
  VAR
    rTrim : REAL;
  END_VAR

            (* FB_XLineTrack — X 直行按航向误差纠偏差速 / 原地左右转。
   eMode: 0=无  1=直行(rBaseVel 带符号 + 纠偏)  2=左旋  3=右旋 *)

rTrim := LIMIT(-ABS(rTrimMax), rKpTrack * rHeadingErr, ABS(rTrimMax));

CASE eMode OF
    1:
        rVelM1 := rBaseVel + rTrim;
        rVelM2 := rBaseVel - rTrim;
    2:
        rVelM1 := ABS(rSpinVel);
        rVelM2 := -ABS(rSpinVel);
    3:
        rVelM1 := -ABS(rSpinVel);
        rVelM2 := ABS(rSpinVel);
ELSE
    rVelM1 := 0.0;
    rVelM2 := 0.0;
END_CASE;

IF xStop OR NOT xEnable THEN
    rVelM1 := 0.0;
    rVelM2 := 0.0;
END_IF;

xActive := (eMode <> 0) AND xEnable AND NOT xStop;
          
END_FUNCTION_BLOCK

FUNCTION_BLOCK FB_ForceFollow
  VAR_INPUT
    rForceSet : REAL;  (* 目标力 N *)
    rForceAct : REAL;  (* 实际力 N *)
    rKp : REAL;  (* 比例增益，越大响应越快，过大易抖 *)
    rVelMax : REAL;  (* 速度限幅（正值） *)
    rDeadband : REAL;  (* 死区 N，区内输出 0 *)
    rPosZ : LREAL;  (* Z 实际位置 *)
    rLimPos : REAL;  (* Z 正限位（同 Cfg_rLimZPos） *)
    rLimNeg : REAL;  (* Z 负限位（同 Cfg_rLimZNeg） *)
    xEnable : BOOL;  (* 力跟随使能（电平） *)
    xInvert : BOOL;  (* 现场方向翻转 *)
  END_VAR
  VAR_OUTPUT
    rZVelCmd : REAL;  (* Z 速度指令输出 *)
    xInBand : BOOL;  (* 力在死区内 *)
  END_VAR
  VAR
    rErr : REAL;
    rV : REAL;
  END_VAR

            (* FB_ForceFollow — Z 恒力 P 控制律；向下=负增压；硬限位 [rLimNeg, rLimPos] 内跟随 *)

IF NOT xEnable THEN
    rZVelCmd := 0.0;
    xInBand := FALSE;
    RETURN;
END_IF;

rErr := rForceSet - rForceAct;
rV := -rKp * rErr;
IF xInvert THEN
    rV := -rV;
END_IF;
rV := LIMIT(-ABS(rVelMax), rV, ABS(rVelMax));

xInBand := ABS(rErr) < rDeadband;
IF xInBand THEN
    rV := 0.0;
END_IF;

(* 硬限位：越限方向输出 0（FB_Servo 另有最终闸门） *)
IF (rPosZ >= rLimPos) AND (rV > 0.0) THEN
    rV := 0.0;
END_IF;
IF (rPosZ <= rLimNeg) AND (rV < 0.0) THEN
    rV := 0.0;
END_IF;

rZVelCmd := rV;
          
END_FUNCTION_BLOCK

FUNCTION_BLOCK FB_Force
  VAR_INPUT
    wRaw : WORD;  (* 组态映射原始力 %IW102 *)
    rScale : REAL;  (* 倍率，默认 0.01 *)
    xEnable : BOOL;  (* 通讯总使能 *)
    xTare : BOOL;  (* 去皮（上升沿记偏移） *)
    xUntare : BOOL;  (* 取消去皮（上升沿清偏移） *)
  END_VAR
  VAR_OUTPUT
    rForceN : REAL;  (* 实际力 N *)
    iRaw : INT;  (* 有符号原始计数 *)
    xCommOk : BOOL;  (* 通讯正常 *)
    xTimeout : BOOL;  (* 2s 原始值不变 → 超时（报警 1005） *)
  END_VAR
  VAR
    rTare : REAL;
    xTarePrev : BOOL;
    xUntarePrev : BOOL;
    wPrev : WORD;
    tonStale : TON;
    rRawScaled : REAL;
  END_VAR

            (* FB_Force — Modbus 原始力换算 + 软件去皮 + 通讯看门狗（仅提示，不进故障） *)

iRaw := WORD_TO_INT(wRaw);
rRawScaled := INT_TO_REAL(iRaw) * rScale;

IF xTare AND NOT xTarePrev THEN
    rTare := rRawScaled;
END_IF;
xTarePrev := xTare;
IF xUntare AND NOT xUntarePrev THEN
    rTare := 0.0;
END_IF;
xUntarePrev := xUntare;

rForceN := rRawScaled - rTare;

tonStale(IN := xEnable AND (wRaw = wPrev), PT := T#2S);
wPrev := wRaw;
xTimeout := xEnable AND tonStale.Q;
xCommOk := xEnable AND NOT xTimeout;
          
END_FUNCTION_BLOCK

FUNCTION_BLOCK FB_Servo
  VAR_INPUT
    xEnable : BOOL;  (* 驱动器使能（来自 AxisCmd_xPower） *)
    xStop : BOOL;  (* 停止运动（保持使能） *)
    xResetFault : BOOL;  (* 故障复位（上升沿） *)
    xHome : BOOL;  (* 回零（电平，完成/撤销后由上层清） *)
    xMoveAbs : BOOL;  (* 绝对定位（电平保持至完成） *)
    rTargetPos : REAL;  (* 绝对目标位置 *)
    xMoveRel : BOOL;  (* 相对定位（电平保持至完成） *)
    rDist : REAL;  (* 相对距离（可正可负） *)
    xUseVelCmd : BOOL;  (* 速度指令模式（力跟随/X双驱） *)
    rVelCmd : REAL;  (* 速度给定（可正可负；|v|<1e-6 视为撤销） *)
    xJogPos : BOOL;  (* 点动+（电平，MC_Jog） *)
    xJogNeg : BOOL;  (* 点动-（电平，MC_Jog） *)
    rJogVel : REAL;  (* 点动速度（正值） *)
    rVel : REAL;  (* 定位速度（正值） *)
    rAcc : REAL;  (* 加速度 *)
    rDec : REAL;  (* 减速度 *)
    xLimEn : BOOL;  (* 硬限位使能（X=FALSE，Y/Z/R=TRUE） *)
    rLimPos : REAL;  (* 正方向硬限位（可手动改） *)
    rLimNeg : REAL;  (* 负方向硬限位（可手动改） *)
  END_VAR
  VAR_OUTPUT
    xPowered : BOOL;  (* 驱动器已上电 := fbPower.Status *)
    xReady : BOOL;  (* 就绪 := 上电且无故障 *)
    xMoving : BOOL;  (* 运动中（含回零） *)
    xStandstill : BOOL;  (* 静止 *)
    xHomed : BOOL;  (* 回零完成（置零后保持） *)
    xFault : BOOL;  (* 故障 := MC_ReadStatus.ErrorStop *)
    xMoveRelDone : BOOL;  (* 相对定位完成 *)
    xMoveAbsDone : BOOL;  (* 绝对定位完成 *)
    rActPos : LREAL;  (* 实际位置 *)
    xVelReq : BOOL;  (* 诊断：仲裁后速度请求已成立 *)
    xVelBusy : BOOL;  (* 诊断：MC_MoveVelocity.Busy *)
    xVelInVel : BOOL;  (* 诊断：MC_MoveVelocity.InVelocity *)
    xErrPower : BOOL;  (* 诊断：MC_Power.Error（驱动未就绪/通讯异常） *)
    xErrVel : BOOL;  (* 诊断：MC_MoveVelocity.Error（参数/平台拒绝） *)
    xErrJog : BOOL;  (* 诊断：MC_Jog.Error *)
    xErrHalt : BOOL;  (* 诊断：MC_Halt.Error *)
    xErrHome : BOOL;  (* 诊断：MC_Home.Error *)
    xErrAbs : BOOL;  (* 诊断：MC_MoveAbsolute.Error *)
    xErrRel : BOOL;  (* 诊断：MC_MoveRelative.Error *)
  END_VAR
  VAR
    fbPower : MC_Power;
    fbHalt : MC_Halt;
    fbHome : MC_Home;
    fbReset : MC_Reset;
    fbReadStatus : MC_ReadStatus;
    fbReadPos : MC_ReadActualPosition;
    fbSetPos : MC_SetPosition;
    fbMoveRel : MC_MoveRelative;
    fbMoveAbs : MC_MoveAbsolute;
    fbMoveVel : MC_MoveVelocity;
    fbJog : MC_Jog;
    eDir : MC_DIRECTION;
    xReqStop : BOOL;
    xReqHome : BOOL;
    xReqAbs : BOOL;
    xReqRel : BOOL;
    xReqVel : BOOL;
    xReqJogPos : BOOL;
    xReqJogNeg : BOOL;
    xReqAny : BOOL;
    xReqHomePrev : BOOL;
    xSetZeroTrig : BOOL;
    xVelRunPrev : BOOL;
    xDirFlip : BOOL;
    xNeedStop : BOOL;
    xHaltPrev : BOOL;
    xResetPrev : BOOL;
    xBlockPos : BOOL;
    xBlockNeg : BOOL;
    rAbsTarget : REAL;
    rRelDist : REAL;
    rVelInPrev : REAL;
  END_VAR
  VAR_IN_OUT
    Axis : AXIS_REF_SM3;
  END_VAR

            (* =============================================================================
   FB_Servo — 单轴原子封装（SM3_Basic）。仅在 PRG_Axis_Control 任务内实例化。

   仲裁优先级：停止/故障 > 回零 > 绝对定位 > 相对定位 > 速度指令 > 点动。
   - 手动点动走 MC_Jog（松开即减速停）；速度指令走 MC_MoveVelocity
   - 运动切换靠 PLCopen 中止机制（新命令 FB 上升沿自动 abort 旧运动）
   - 全部运动请求撤销（松手/速度归零/停止/急停/撞限位）→ MC_Halt 减速停车
   - 硬限位：xLimEn=TRUE 时，所有模式都限制在 [rLimNeg, rLimPos] 内：
     点动/速度 越限方向被禁止；定位目标被夹紧；X 轴传 xLimEn:=FALSE
   ========================================================================== *)

(* 1. 状态与位置 *)
fbReadStatus(Axis := Axis, Enable := TRUE);
fbReadPos(Axis := Axis, Enable := TRUE);
rActPos := fbReadPos.Position;
xStandstill := fbReadStatus.StandStill;
xFault := fbReadStatus.ErrorStop;
xMoving := fbReadStatus.DiscreteMotion OR fbReadStatus.ContinuousMotion OR fbReadStatus.Homing;

(* 2. 故障复位（上升沿） *)
fbReset(Axis := Axis, Execute := xResetFault AND NOT xResetPrev);
xResetPrev := xResetFault;

(* 3. 驱动器使能（xStop 不掉使能） *)
fbPower(Axis := Axis, Enable := TRUE,
        bRegulatorOn := xEnable AND NOT xFault,
        bDriveStart := xEnable AND NOT xFault);
xPowered := fbPower.Status;
xReady := xPowered AND NOT xFault;

(* 4. 硬限位：越限方向禁止；定位目标夹紧（已越限时仍允许向回运动） *)
xBlockPos := xLimEn AND (rActPos >= rLimPos);
xBlockNeg := xLimEn AND (rActPos <= rLimNeg);
rAbsTarget := rTargetPos;
rRelDist := rDist;
IF xLimEn THEN
    rAbsTarget := LIMIT(rLimNeg, rTargetPos, rLimPos);
    rRelDist := LIMIT(rLimNeg, rActPos + rDist, rLimPos) - rActPos;
END_IF;

(* 5. 命令仲裁：停止/故障 > 回零 > 绝对 > 相对 > 速度 > 点动 *)
xReqStop := xStop OR NOT xEnable OR xFault;
xReqHome := xHome AND NOT xReqStop;
xReqAbs := xMoveAbs AND xPowered AND NOT xReqStop AND NOT xReqHome;
xReqRel := xMoveRel AND (ABS(rRelDist) > 1.0E-9) AND xPowered
           AND NOT xReqStop AND NOT xReqHome AND NOT xReqAbs;
xReqVel := xUseVelCmd AND (ABS(rVelCmd) > 1.0E-6) AND xPowered
           AND NOT ((rVelCmd > 0.0) AND xBlockPos) AND NOT ((rVelCmd < 0.0) AND xBlockNeg)
           AND NOT xReqStop AND NOT xReqHome AND NOT xReqAbs AND NOT xReqRel;
xReqJogPos := xJogPos AND NOT xJogNeg AND NOT xBlockPos AND xPowered
              AND NOT xReqStop AND NOT xReqHome AND NOT xReqAbs AND NOT xReqRel AND NOT xReqVel;
xReqJogNeg := xJogNeg AND NOT xJogPos AND NOT xBlockNeg AND xPowered
              AND NOT xReqStop AND NOT xReqHome AND NOT xReqAbs AND NOT xReqRel AND NOT xReqVel;
xReqAny := xReqHome OR xReqAbs OR xReqRel OR xReqVel OR xReqJogPos OR xReqJogNeg;

(* 6. 回零：MC_Home(0) → MC_SetPosition(0) → xHomed *)
IF xReqHome AND NOT xReqHomePrev THEN
    xHomed := FALSE;
END_IF;
xReqHomePrev := xReqHome;
fbHome(Axis := Axis, Execute := xReqHome, Position := 0.0);
IF fbHome.Done THEN
    xSetZeroTrig := TRUE;
END_IF;
fbSetPos(Axis := Axis, Execute := xSetZeroTrig, Position := 0.0);
IF fbSetPos.Done THEN
    xHomed := TRUE;
    xSetZeroTrig := FALSE;
END_IF;

(* 7. 绝对 / 相对定位（目标已夹紧；电平保持 Execute，Done 上报） *)
fbMoveAbs(Axis := Axis, Execute := xReqAbs, Position := rAbsTarget,
          Velocity := ABS(rVel), Acceleration := rAcc, Deceleration := rDec);
fbMoveRel(Axis := Axis, Execute := xReqRel, Distance := rRelDist,
          Velocity := ABS(rVel), Acceleration := rAcc, Deceleration := rDec);
xMoveAbsDone := fbMoveAbs.Done;
xMoveRelDone := fbMoveRel.Done;

(* 8. 速度指令：MC_MoveVelocity；Velocity 取绝对值，方向走 Direction *)
(* 注意：本机 SM3 库的方向字面值是 positive/negative（非 CoDeSys 的 mcPositiveDirection） *)
IF rVelCmd >= 0.0 THEN
    eDir := positive;
ELSE
    eDir := negative;
END_IF;
(* 运行中换向：先撤 Execute 一拍，下一拍带新方向重新触发 *)
xDirFlip := xReqVel AND xVelRunPrev AND ((rVelCmd >= 0.0) <> (rVelInPrev >= 0.0));
fbMoveVel(Axis := Axis, Execute := xReqVel AND NOT xDirFlip,
          Velocity := ABS(rVelCmd), Direction := eDir,
          Acceleration := rAcc, Deceleration := rDec);
xVelRunPrev := xReqVel;
rVelInPrev := rVelCmd;

(* 9. 手动点动：MC_Jog（按住动、松开减速停；越限方向已在仲裁禁止） *)
fbJog(Axis := Axis,
      JogForward := xReqJogPos,
      JogBackward := xReqJogNeg,
      Velocity := ABS(rJogVel),
      Acceleration := rAcc,
      Deceleration := rDec);

(* 10. 停车：有使能但无任何运动请求（松手/速度归零/停止/急停/撞限位）→ MC_Halt *)
xNeedStop := xPowered AND NOT xReqAny;
fbHalt(Axis := Axis, Execute := xNeedStop AND xMoving AND NOT xHaltPrev,
       Deceleration := rDec);
xHaltPrev := xNeedStop AND xMoving;

(* 11. 诊断输出（g 线 0.5） *)
xVelReq := xReqVel;
xVelBusy := fbMoveVel.Busy;
xVelInVel := fbMoveVel.InVelocity;
xErrPower := fbPower.Error;
xErrVel := fbMoveVel.Error;
xErrJog := fbJog.Error;
xErrHalt := fbHalt.Error;
xErrHome := fbHome.Error;
xErrAbs := fbMoveAbs.Error;
xErrRel := fbMoveRel.Error;
          
END_FUNCTION_BLOCK

PROGRAM PRG_TcpHmi
  VAR
    xInit : BOOL;
    xPanelOp : BOOL;
    xTcpOp : BOOL;
    xValid : BOOL;
    wMagic : WORD;
    wVersion : WORD;
    wSeqHead : WORD;
    wSeqTail : WORD;
    wHeartbeat : WORD;
    dwTmp : DWORD;
    diTmp : DINT;
    i : INT;
    tonHb : TON;
  END_VAR

            (* PRG_TcpHmi — Modbus TCP 过程映像编解码 + 控制源仲裁。
   PLC=Master 读 Holding1000 / 写 Holding1100；Gateway=Server。
   eCtrlSrc 为 GVL 变量：0=面板/触摸屏 1=远程(Web)。 *)

IF NOT xInit THEN
    Tcp_xEStop := TRUE;
    Tcp_rJogVelX := 0.4; Tcp_rSpinVel := 0.3;
    Tcp_rJogVelY := 0.3; Tcp_rJogVelZ := 0.2; Tcp_rJogVelR := 0.2;
    Tcp_rAutoDistX := 1.0; Tcp_rAutoVelX := 0.4;
    Tcp_rAutoVelY := 0.3; Tcp_rAutoVelZ := 0.15;
    Tcp_rWheelBase := 5.0; Tcp_rForceSet := 100.0;
    Tcp_xForceSimEnable := FALSE;
    Tcp_iAutoPasses := 1;
    Tcp_rHeadingErr := 0.0;
    Tcp_rKpTrack := 0.0; Tcp_rKpForce := 1.0;
    Tcp_rAccX := 100.0; Tcp_rDecX := 100.0;
    Tcp_rAccY := 100.0; Tcp_rDecY := 100.0;
    Tcp_rAccZ := 100.0; Tcp_rDecZ := 100.0;
    Tcp_rAccR := 100.0; Tcp_rDecR := 100.0;
    Tcp_iCommStatus := 0;
    Tcp_wLastHb := 0; Tcp_wLastSeq := 16#FFFF; Tcp_wStatusSeq := 0;
    tonHb(IN := FALSE);
    xInit := TRUE;
END_IF;

(* ===== 命令快照解码 ===== *)
wMagic := MB_CmdIn[0];
wVersion := MB_CmdIn[1];
wSeqHead := MB_CmdIn[2];
wHeartbeat := MB_CmdIn[3];
wSeqTail := MB_CmdIn[63];
xValid := (wMagic = 19533) AND (wVersion = 256) AND (wSeqHead = wSeqTail);
IF xValid THEN
    Tcp_iCommStatus := 1;
    IF wHeartbeat <> Tcp_wLastHb THEN
        tonHb(IN := FALSE);
        tonHb(IN := TRUE, PT := T#1S);
        Tcp_wLastHb := wHeartbeat;
    END_IF;
    IF wSeqHead <> Tcp_wLastSeq THEN
        Tcp_wLastSeq := wSeqHead;
        Tcp_xEStop := (MB_CmdIn[4] AND 1) <> 0;
        Tcp_xStop := (MB_CmdIn[4] AND 2) <> 0;
        Tcp_xStopHold3s := (MB_CmdIn[4] AND 4) <> 0;
        Tcp_xStart := (MB_CmdIn[4] AND 8) <> 0;
        Tcp_xEnable := (MB_CmdIn[4] AND 16) <> 0;
        Tcp_xAutoMode := (MB_CmdIn[4] AND 32) <> 0;
        Tcp_xJogXPos := (MB_CmdIn[4] AND 64) <> 0;
        Tcp_xJogXNeg := (MB_CmdIn[4] AND 128) <> 0;
        Tcp_xSpinLeft := (MB_CmdIn[4] AND 256) <> 0;
        Tcp_xSpinRight := (MB_CmdIn[4] AND 512) <> 0;
        Tcp_xJogYPos := (MB_CmdIn[4] AND 1024) <> 0;
        Tcp_xJogYNeg := (MB_CmdIn[4] AND 2048) <> 0;
        Tcp_xJogZPos := (MB_CmdIn[4] AND 4096) <> 0;
        Tcp_xJogZNeg := (MB_CmdIn[4] AND 8192) <> 0;
        Tcp_xJogRPos := (MB_CmdIn[4] AND 16384) <> 0;
        Tcp_xJogRNeg := (MB_CmdIn[4] AND 32768) <> 0;
        Tcp_xHomeY := (MB_CmdIn[5] AND 1) <> 0;
        Tcp_xHomeZ := (MB_CmdIn[5] AND 2) <> 0;
        Tcp_xHomeR := (MB_CmdIn[5] AND 4) <> 0;
        Tcp_xHomeExec := (MB_CmdIn[5] AND 8) <> 0;
        Tcp_xAutoStart := (MB_CmdIn[5] AND 16) <> 0;
        Tcp_xAutoAbort := (MB_CmdIn[5] AND 32) <> 0;
        Tcp_xForceSimEnable := (MB_CmdIn[5] AND 64) <> 0;
        Tcp_xForceTare := (MB_CmdIn[5] AND 128) <> 0;
        Tcp_xForceUntare := (MB_CmdIn[5] AND 256) <> 0;
        Tcp_xForceGuide := (MB_CmdIn[5] AND 512) <> 0;
        Tcp_iHomeAxis := WORD_TO_INT(MB_CmdIn[6]);
        Tcp_iAutoPasses := WORD_TO_INT(MB_CmdIn[7]);
        dwTmp := SHL(WORD_TO_DWORD(MB_CmdIn[8]), 16) OR WORD_TO_DWORD(MB_CmdIn[9]);
        Tcp_rJogVelX := DINT_TO_REAL(DWORD_TO_DINT(dwTmp)) / 1000.0;
        dwTmp := SHL(WORD_TO_DWORD(MB_CmdIn[10]), 16) OR WORD_TO_DWORD(MB_CmdIn[11]);
        Tcp_rSpinVel := DINT_TO_REAL(DWORD_TO_DINT(dwTmp)) / 1000.0;
        dwTmp := SHL(WORD_TO_DWORD(MB_CmdIn[12]), 16) OR WORD_TO_DWORD(MB_CmdIn[13]);
        Tcp_rJogVelY := DINT_TO_REAL(DWORD_TO_DINT(dwTmp)) / 1000.0;
        dwTmp := SHL(WORD_TO_DWORD(MB_CmdIn[14]), 16) OR WORD_TO_DWORD(MB_CmdIn[15]);
        Tcp_rJogVelZ := DINT_TO_REAL(DWORD_TO_DINT(dwTmp)) / 1000.0;
        dwTmp := SHL(WORD_TO_DWORD(MB_CmdIn[16]), 16) OR WORD_TO_DWORD(MB_CmdIn[17]);
        Tcp_rJogVelR := DINT_TO_REAL(DWORD_TO_DINT(dwTmp)) / 1000.0;
        dwTmp := SHL(WORD_TO_DWORD(MB_CmdIn[18]), 16) OR WORD_TO_DWORD(MB_CmdIn[19]);
        Tcp_rAutoDistX := DINT_TO_REAL(DWORD_TO_DINT(dwTmp)) / 1000.0;
        dwTmp := SHL(WORD_TO_DWORD(MB_CmdIn[20]), 16) OR WORD_TO_DWORD(MB_CmdIn[21]);
        Tcp_rAutoVelX := DINT_TO_REAL(DWORD_TO_DINT(dwTmp)) / 1000.0;
        dwTmp := SHL(WORD_TO_DWORD(MB_CmdIn[22]), 16) OR WORD_TO_DWORD(MB_CmdIn[23]);
        Tcp_rAutoVelY := DINT_TO_REAL(DWORD_TO_DINT(dwTmp)) / 1000.0;
        dwTmp := SHL(WORD_TO_DWORD(MB_CmdIn[24]), 16) OR WORD_TO_DWORD(MB_CmdIn[25]);
        Tcp_rAutoVelZ := DINT_TO_REAL(DWORD_TO_DINT(dwTmp)) / 1000.0;
        dwTmp := SHL(WORD_TO_DWORD(MB_CmdIn[26]), 16) OR WORD_TO_DWORD(MB_CmdIn[27]);
        Tcp_rWheelBase := DINT_TO_REAL(DWORD_TO_DINT(dwTmp)) / 1000.0;
        dwTmp := SHL(WORD_TO_DWORD(MB_CmdIn[28]), 16) OR WORD_TO_DWORD(MB_CmdIn[29]);
        Tcp_rForceSet := DINT_TO_REAL(DWORD_TO_DINT(dwTmp)) / 100.0;
        dwTmp := SHL(WORD_TO_DWORD(MB_CmdIn[30]), 16) OR WORD_TO_DWORD(MB_CmdIn[31]);
        Tcp_rForceSim := DINT_TO_REAL(DWORD_TO_DINT(dwTmp)) / 100.0;
        dwTmp := SHL(WORD_TO_DWORD(MB_CmdIn[32]), 16) OR WORD_TO_DWORD(MB_CmdIn[33]);
        Tcp_rHeadingErr := DINT_TO_REAL(DWORD_TO_DINT(dwTmp)) / 1000.0;
        dwTmp := SHL(WORD_TO_DWORD(MB_CmdIn[34]), 16) OR WORD_TO_DWORD(MB_CmdIn[35]);
        Tcp_rKpTrack := DINT_TO_REAL(DWORD_TO_DINT(dwTmp)) / 1000.0;
        dwTmp := SHL(WORD_TO_DWORD(MB_CmdIn[36]), 16) OR WORD_TO_DWORD(MB_CmdIn[37]);
        Tcp_rKpForce := DINT_TO_REAL(DWORD_TO_DINT(dwTmp)) / 1000.0;
        dwTmp := SHL(WORD_TO_DWORD(MB_CmdIn[38]), 16) OR WORD_TO_DWORD(MB_CmdIn[39]);
        Tcp_rAccX := DINT_TO_REAL(DWORD_TO_DINT(dwTmp)) / 1000.0;
        dwTmp := SHL(WORD_TO_DWORD(MB_CmdIn[40]), 16) OR WORD_TO_DWORD(MB_CmdIn[41]);
        Tcp_rDecX := DINT_TO_REAL(DWORD_TO_DINT(dwTmp)) / 1000.0;
        dwTmp := SHL(WORD_TO_DWORD(MB_CmdIn[42]), 16) OR WORD_TO_DWORD(MB_CmdIn[43]);
        Tcp_rAccY := DINT_TO_REAL(DWORD_TO_DINT(dwTmp)) / 1000.0;
        dwTmp := SHL(WORD_TO_DWORD(MB_CmdIn[44]), 16) OR WORD_TO_DWORD(MB_CmdIn[45]);
        Tcp_rDecY := DINT_TO_REAL(DWORD_TO_DINT(dwTmp)) / 1000.0;
        dwTmp := SHL(WORD_TO_DWORD(MB_CmdIn[46]), 16) OR WORD_TO_DWORD(MB_CmdIn[47]);
        Tcp_rAccZ := DINT_TO_REAL(DWORD_TO_DINT(dwTmp)) / 1000.0;
        dwTmp := SHL(WORD_TO_DWORD(MB_CmdIn[48]), 16) OR WORD_TO_DWORD(MB_CmdIn[49]);
        Tcp_rDecZ := DINT_TO_REAL(DWORD_TO_DINT(dwTmp)) / 1000.0;
        dwTmp := SHL(WORD_TO_DWORD(MB_CmdIn[50]), 16) OR WORD_TO_DWORD(MB_CmdIn[51]);
        Tcp_rAccR := DINT_TO_REAL(DWORD_TO_DINT(dwTmp)) / 1000.0;
        dwTmp := SHL(WORD_TO_DWORD(MB_CmdIn[52]), 16) OR WORD_TO_DWORD(MB_CmdIn[53]);
        Tcp_rDecR := DINT_TO_REAL(DWORD_TO_DINT(dwTmp)) / 1000.0;
    END_IF;
ELSIF wMagic <> 0 AND wMagic <> 19533 THEN
    Tcp_iCommStatus := 2;
ELSIF wSeqHead <> wSeqTail THEN
    Tcp_iCommStatus := 3;
END_IF;
tonHb();
IF tonHb.Q OR Tcp_iCommStatus = 0 THEN
    Tcp_xTimeout := TRUE;
    Tcp_xConnected := FALSE;
    Tcp_xOnline := FALSE;
    IF tonHb.Q THEN Tcp_iCommStatus := 4; END_IF;
    Tcp_xJogXPos := FALSE; Tcp_xJogXNeg := FALSE;
    Tcp_xSpinLeft := FALSE; Tcp_xSpinRight := FALSE;
    Tcp_xJogYPos := FALSE; Tcp_xJogYNeg := FALSE;
    Tcp_xJogZPos := FALSE; Tcp_xJogZNeg := FALSE;
    Tcp_xJogRPos := FALSE; Tcp_xJogRNeg := FALSE;
    Tcp_xHomeY := FALSE; Tcp_xHomeZ := FALSE; Tcp_xHomeR := FALSE;
    Tcp_xHomeExec := FALSE;
    Tcp_xStart := FALSE; Tcp_xEnable := FALSE;
    Tcp_xAutoStart := FALSE;
    Tcp_xForceTare := FALSE; Tcp_xForceUntare := FALSE; Tcp_xForceGuide := FALSE;
    Tcp_xStop := TRUE;
    Tcp_xAutoAbort := TRUE;
    Tcp_xEStop := TRUE;
ELSE
    Tcp_xTimeout := FALSE;
    Tcp_xConnected := TRUE;
    Tcp_xOnline := TRUE;
END_IF;

(* ===== 状态快照编码 ===== *)
Tcp_wStatusSeq := Tcp_wStatusSeq + 1;
MB_StatusOut[0] := 19533;
MB_StatusOut[1] := 256;
MB_StatusOut[2] := Tcp_wStatusSeq;
MB_StatusOut[3] := Tcp_wLastSeq;
MB_StatusOut[4] := Tcp_wLastHb;
FOR i := 5 TO 62 DO MB_StatusOut[i] := 0; END_FOR;
MB_StatusOut[5] := INT_TO_WORD(Tcp_iCommStatus);
MB_StatusOut[6] := INT_TO_WORD(HMI_eDevState);
MB_StatusOut[7] := INT_TO_WORD(HMI_eOpMode);
MB_StatusOut[8] := INT_TO_WORD(HMI_iAlarmShow);
MB_StatusOut[9] := INT_TO_WORD(HMI_iAutoStepShow);
IF HMI_xDevStop THEN MB_StatusOut[10] := MB_StatusOut[10] OR 1; END_IF;
IF HMI_xDevRun THEN MB_StatusOut[10] := MB_StatusOut[10] OR 2; END_IF;
IF HMI_xDevError THEN MB_StatusOut[10] := MB_StatusOut[10] OR 4; END_IF;
IF HMI_xLampEStop THEN MB_StatusOut[10] := MB_StatusOut[10] OR 8; END_IF;
IF HMI_xLampEnableOk THEN MB_StatusOut[10] := MB_StatusOut[10] OR 16; END_IF;
IF HMI_xLampFault THEN MB_StatusOut[10] := MB_StatusOut[10] OR 32; END_IF;
IF HMI_xAutoBusy THEN MB_StatusOut[10] := MB_StatusOut[10] OR 64; END_IF;
IF HMI_xAutoDone THEN MB_StatusOut[10] := MB_StatusOut[10] OR 128; END_IF;
IF HMI_xHomedY THEN MB_StatusOut[10] := MB_StatusOut[10] OR 256; END_IF;
IF HMI_xHomedZ THEN MB_StatusOut[10] := MB_StatusOut[10] OR 512; END_IF;
IF HMI_xHomedR THEN MB_StatusOut[10] := MB_StatusOut[10] OR 1024; END_IF;
IF HMI_xHomeBusyY THEN MB_StatusOut[10] := MB_StatusOut[10] OR 2048; END_IF;
IF HMI_xHomeBusyZ THEN MB_StatusOut[10] := MB_StatusOut[10] OR 4096; END_IF;
IF HMI_xHomeBusyR THEN MB_StatusOut[10] := MB_StatusOut[10] OR 8192; END_IF;
IF Tcp_xConnected THEN MB_StatusOut[10] := MB_StatusOut[10] OR 16384; END_IF;
IF Tcp_xTimeout THEN MB_StatusOut[10] := MB_StatusOut[10] OR 32768; END_IF;
IF Force_xCommOk THEN MB_StatusOut[11] := MB_StatusOut[11] OR 1; END_IF;
IF Force_xTimeout THEN MB_StatusOut[11] := MB_StatusOut[11] OR 2; END_IF;
IF Force_xSlaveFail THEN MB_StatusOut[11] := MB_StatusOut[11] OR 4; END_IF;
IF Force_xTareBusy THEN MB_StatusOut[11] := MB_StatusOut[11] OR 8; END_IF;
IF Force_xTareDone THEN MB_StatusOut[11] := MB_StatusOut[11] OR 16; END_IF;
IF AxisFb_xReady THEN MB_StatusOut[11] := MB_StatusOut[11] OR 32; END_IF;
IF AxisFb_xMoveDoneX THEN MB_StatusOut[11] := MB_StatusOut[11] OR 64; END_IF;
IF AxisFb_xMoveDoneY THEN MB_StatusOut[11] := MB_StatusOut[11] OR 128; END_IF;
IF AxisFb_xFaultM1 THEN MB_StatusOut[11] := MB_StatusOut[11] OR 256; END_IF;
IF AxisFb_xFaultM2 THEN MB_StatusOut[11] := MB_StatusOut[11] OR 512; END_IF;
IF AxisFb_xFaultY THEN MB_StatusOut[11] := MB_StatusOut[11] OR 1024; END_IF;
IF AxisFb_xFaultZ THEN MB_StatusOut[11] := MB_StatusOut[11] OR 2048; END_IF;
IF AxisFb_xFaultR THEN MB_StatusOut[11] := MB_StatusOut[11] OR 4096; END_IF;
IF AxisFb_xHomedY THEN MB_StatusOut[11] := MB_StatusOut[11] OR 8192; END_IF;
IF AxisFb_xHomedZ THEN MB_StatusOut[11] := MB_StatusOut[11] OR 16384; END_IF;
IF AxisFb_xHomedR THEN MB_StatusOut[11] := MB_StatusOut[11] OR 32768; END_IF;
diTmp := REAL_TO_DINT(HMI_rForceShow * 100.0);
dwTmp := DINT_TO_DWORD(diTmp);
MB_StatusOut[12] := DWORD_TO_WORD(SHR(dwTmp, 16));
MB_StatusOut[13] := DWORD_TO_WORD(dwTmp AND 16#FFFF);
diTmp := REAL_TO_DINT(AxisFb_rPosM1 * 1000.0);
dwTmp := DINT_TO_DWORD(diTmp);
MB_StatusOut[14] := DWORD_TO_WORD(SHR(dwTmp, 16));
MB_StatusOut[15] := DWORD_TO_WORD(dwTmp AND 16#FFFF);
diTmp := REAL_TO_DINT(AxisFb_rPosM2 * 1000.0);
dwTmp := DINT_TO_DWORD(diTmp);
MB_StatusOut[16] := DWORD_TO_WORD(SHR(dwTmp, 16));
MB_StatusOut[17] := DWORD_TO_WORD(dwTmp AND 16#FFFF);
diTmp := REAL_TO_DINT(AxisFb_rPosY * 1000.0);
dwTmp := DINT_TO_DWORD(diTmp);
MB_StatusOut[18] := DWORD_TO_WORD(SHR(dwTmp, 16));
MB_StatusOut[19] := DWORD_TO_WORD(dwTmp AND 16#FFFF);
diTmp := REAL_TO_DINT(AxisFb_rPosZ * 1000.0);
dwTmp := DINT_TO_DWORD(diTmp);
MB_StatusOut[20] := DWORD_TO_WORD(SHR(dwTmp, 16));
MB_StatusOut[21] := DWORD_TO_WORD(dwTmp AND 16#FFFF);
diTmp := REAL_TO_DINT(AxisFb_rPosR * 1000.0);
dwTmp := DINT_TO_DWORD(diTmp);
MB_StatusOut[22] := DWORD_TO_WORD(SHR(dwTmp, 16));
MB_StatusOut[23] := DWORD_TO_WORD(dwTmp AND 16#FFFF);
diTmp := REAL_TO_DINT(AxisFb_rVelCmdM1 * 1000.0);
dwTmp := DINT_TO_DWORD(diTmp);
MB_StatusOut[24] := DWORD_TO_WORD(SHR(dwTmp, 16));
MB_StatusOut[25] := DWORD_TO_WORD(dwTmp AND 16#FFFF);
diTmp := REAL_TO_DINT(AxisFb_rVelCmdM2 * 1000.0);
dwTmp := DINT_TO_DWORD(diTmp);
MB_StatusOut[26] := DWORD_TO_WORD(SHR(dwTmp, 16));
MB_StatusOut[27] := DWORD_TO_WORD(dwTmp AND 16#FFFF);
MB_StatusOut[63] := Tcp_wStatusSeq;

(* ===== 控制源仲裁 ===== *)
xPanelOp := StartBtn OR StopBtn OR ResetBtn OR JogFwd OR JogBwd OR JogLeft OR JogRight
    OR JogUp OR JogDown OR JogClockAdd OR JogClockMis;
xTcpOp := Tcp_xOnline AND (
    Tcp_xStart OR Tcp_xStop OR Tcp_xStopHold3s OR Tcp_xAutoStart OR Tcp_xAutoAbort
    OR Tcp_xJogXPos OR Tcp_xJogXNeg OR Tcp_xSpinLeft OR Tcp_xSpinRight
    OR Tcp_xJogYPos OR Tcp_xJogYNeg OR Tcp_xJogZPos OR Tcp_xJogZNeg
    OR Tcp_xJogRPos OR Tcp_xJogRNeg
    OR Tcp_xHomeY OR Tcp_xHomeZ OR Tcp_xHomeR OR Tcp_xHomeExec
    OR Tcp_xForceGuide OR Tcp_xForceTare OR Tcp_xForceUntare);
IF NOT Tcp_xOnline THEN
    eCtrlSrc := 0;
ELSIF xTcpOp THEN
    eCtrlSrc := 1;
ELSIF xPanelOp THEN
    eCtrlSrc := 0;
END_IF;

IF eCtrlSrc = 1 THEN
    HMI_xAutoMode := Tcp_xAutoMode;
    HMI_xJogXPos := Tcp_xJogXPos;   HMI_xJogXNeg := Tcp_xJogXNeg;
    HMI_xSpinLeft := Tcp_xSpinLeft; HMI_xSpinRight := Tcp_xSpinRight;
    HMI_xJogYPos := Tcp_xJogYPos;   HMI_xJogYNeg := Tcp_xJogYNeg;
    HMI_xJogZPos := Tcp_xJogZPos;   HMI_xJogZNeg := Tcp_xJogZNeg;
    HMI_xJogRPos := Tcp_xJogRPos;   HMI_xJogRNeg := Tcp_xJogRNeg;
    HMI_xHomeY := Tcp_xHomeY; HMI_xHomeZ := Tcp_xHomeZ; HMI_xHomeR := Tcp_xHomeR;
    HMI_iHomeAxis := Tcp_iHomeAxis; HMI_xHomeExec := Tcp_xHomeExec;
    HMI_xForceGuide := Tcp_xForceGuide;
    HMI_xForceTare := Tcp_xForceTare; HMI_xForceUntare := Tcp_xForceUntare;
    HMI_xForceSimEnable := Tcp_xForceSimEnable;
    HMI_rJogVelX := Tcp_rJogVelX; HMI_rSpinVel := Tcp_rSpinVel;
    HMI_rJogVelY := Tcp_rJogVelY; HMI_rJogVelZ := Tcp_rJogVelZ; HMI_rJogVelR := Tcp_rJogVelR;
    HMI_rAutoDistX := Tcp_rAutoDistX; HMI_rAutoVelX := Tcp_rAutoVelX;
    HMI_rAutoVelY := Tcp_rAutoVelY; HMI_rAutoVelZ := Tcp_rAutoVelZ;
    HMI_rWheelBase := Tcp_rWheelBase; HMI_rForceSet := Tcp_rForceSet;
    HMI_rForceSim := Tcp_rForceSim;
    HMI_iAutoPasses := Tcp_iAutoPasses;
    HMI_rHeadingErr := Tcp_rHeadingErr;
    HMI_rKpTrack := Tcp_rKpTrack;
    HMI_rKpForce := Tcp_rKpForce;
    HMI_rAccX := Tcp_rAccX; HMI_rDecX := Tcp_rDecX;
    HMI_rAccY := Tcp_rAccY; HMI_rDecY := Tcp_rDecY;
    HMI_rAccZ := Tcp_rAccZ; HMI_rDecZ := Tcp_rDecZ;
    HMI_rAccR := Tcp_rAccR; HMI_rDecR := Tcp_rDecR;
END_IF;

HMI_xEStop := EStop AND Tcp_xEStop AND HMI_xEStopReq;
HMI_xStart := StartBtn OR HMI_xStartReq OR (Tcp_xOnline AND Tcp_xStart);
HMI_xEnable := HMI_xStart;
HMI_xStop := StopBtn OR HMI_xStopReq OR (Tcp_xOnline AND Tcp_xStop);
HMI_xStopHold3s := ResetBtn OR HMI_xResetReq OR (Tcp_xOnline AND Tcp_xStopHold3s);
HMI_xAutoStart := (Tcp_xOnline AND Tcp_xAutoStart) OR ((eCtrlSrc = 0) AND HMI_xAutoStartReq);
HMI_xAutoAbort := HMI_xAutoAbortReq OR (Tcp_xOnline AND Tcp_xAutoAbort);
          
END_PROGRAM

PROGRAM PRG_Axis_Control
  VAR
    fbX : FB_XDual;
    fbY : FB_Servo;
    fbZ : FB_Servo;
    fbR : FB_Servo;
    fbForce : FB_Force;
    fbFF : FB_ForceFollow;
  END_VAR

            (* PRG_Axis_Control — 运动独立任务(ETHERCAT 4ms)。只读 AxisCmd_*，写 AxisFb_*/rForceAct。
   禁止被其它 POU CALL；禁止写 HMI_*/报警。
   X：FB_XDual（LineTrack + 双 FB_Servo，无 Virtual/Gear）；Y/Z/R 仍 FB_Servo。 *)

(* ===== 力传感转换（本 POU 拥有 rForceAct） ===== *)
fbForce(wRaw := Force_wInRaw, rScale := Force_rScale, xEnable := Force_xEnable,
    xTare := HMI_xForceTare OR Logic_xForceTare, xUntare := HMI_xForceUntare);
Force_iRaw := fbForce.iRaw;
Force_xCommOk := fbForce.xCommOk;
Force_xTimeout := fbForce.xTimeout;
IF NOT HMI_xForceSimEnable THEN
    rForceAct := fbForce.rForceN;
END_IF;

(* ===== X：FB_XDual（LineTrack + 双 Servo；无 Virtual/Gear） ===== *)
fbX(
    AxisM1 := Axis, AxisM2 := Axis_1,
    xEnable := AxisCmd_xPower, xStop := AxisCmd_xStopAll, xResetFault := AxisCmd_xResetFault,
    xJogPos := AxisCmd_xJogXPos, xJogNeg := AxisCmd_xJogXNeg,
    xSpinLeft := AxisCmd_xSpinLeft, xSpinRight := AxisCmd_xSpinRight,
    xMoveRel := AxisCmd_xMoveRelX, rMoveDist := AxisCmd_rMoveDistX, rMoveVel := AxisCmd_rMoveVelX,
    rJogVel := AxisCmd_rJogVelX, rSpinVel := AxisCmd_rSpinVel,
    rHeadingErr := AxisCmd_rHeadingErr, rKpTrack := AxisCmd_rTrackKp,
    rAcc := AxisCmd_rAccX, rDec := AxisCmd_rDecX,
    rTrimMax := Cfg_rPhaseMax);
AxisFb_xMoveDoneX := fbX.xMoveDone;
AxisFb_rPosX := fbX.rPosV;
AxisFb_rSyncErr := fbX.rSyncErr;
AxisFb_rVelFactorX := fbX.rVelFactor;
AxisFb_xGantryCoupled := fbX.xCoupled;
AxisFb_xInGearM1 := fbX.xInGearM1;
AxisFb_xInGearM2 := fbX.xInGearM2;
AxisFb_xPoweredV := fbX.xPoweredV;
AxisFb_xSyncWarn := fbX.xSyncWarn;
AxisFb_xSyncFault := fbX.xSyncFault;
AxisFb_iGantryState := fbX.iState;
AxisFb_rVelCmdM1 := fbX.rVelCmdM1;
AxisFb_rVelCmdM2 := fbX.rVelCmdM2;
AxisFb_rPosM1 := fbX.rPosM1;
AxisFb_rPosM2 := fbX.rPosM2;
AxisFb_xMovingM1 := fbX.xMovingM1;
AxisFb_xMovingM2 := fbX.xMovingM2;
AxisFb_xStandstill1 := fbX.xStandstillM1;
AxisFb_xStandstill2 := fbX.xStandstillM2;
AxisFb_xPoweredM1 := fbX.xPoweredM1;
AxisFb_xPoweredM2 := fbX.xPoweredM2;
AxisFb_xReadyM1 := fbX.xReadyM1;
AxisFb_xReadyM2 := fbX.xReadyM2;
AxisFb_xFaultM1 := fbX.xFaultM1;
AxisFb_xFaultM2 := fbX.xFaultM2;

(* ===== Y：回零 > 绝对(归位) > 相对(横移) > 点动；硬限位 [Cfg_rLimYNeg, Cfg_rLimYPos] ===== *)
fbY(Axis := Axis_2, xEnable := AxisCmd_xPower, xStop := AxisCmd_xStopAll, xResetFault := AxisCmd_xResetFault,
    xHome := AxisCmd_xHomeY,
    xMoveAbs := AxisCmd_xMoveAbsY, rTargetPos := AxisCmd_rMoveAbsPosY,
    xMoveRel := AxisCmd_xMoveRelY, rDist := AxisCmd_rMoveDistY,
    xJogPos := AxisCmd_xJogYPos, xJogNeg := AxisCmd_xJogYNeg, rJogVel := AxisCmd_rJogVelY,
    rVel := AxisCmd_rMoveVelY, rAcc := AxisCmd_rAccY, rDec := AxisCmd_rDecY,
    xLimEn := TRUE, rLimPos := Cfg_rLimYPos, rLimNeg := Cfg_rLimYNeg);
AxisFb_xMoveDoneY := fbY.xMoveRelDone;

(* ===== Z：力跟随速度 > 回零 > 点动；硬限位 [Cfg_rLimZNeg, Cfg_rLimZPos] ===== *)
fbFF(rForceSet := AxisCmd_rForceSet, rForceAct := rForceAct, rKp := AxisCmd_rForceKp,
    rVelMax := AxisCmd_rForceVelMax, rDeadband := 0.5, rPosZ := fbZ.rActPos,
    rLimPos := Cfg_rLimZPos, rLimNeg := Cfg_rLimZNeg,
    xEnable := AxisCmd_xForceFollow, xInvert := FALSE);
fbZ(Axis := Axis_3, xEnable := AxisCmd_xPower, xStop := AxisCmd_xStopAll, xResetFault := AxisCmd_xResetFault,
    xHome := AxisCmd_xHomeZ,
    xUseVelCmd := AxisCmd_xForceFollow, rVelCmd := fbFF.rZVelCmd,
    xJogPos := AxisCmd_xJogZPos, xJogNeg := AxisCmd_xJogZNeg, rJogVel := AxisCmd_rJogVelZ,
    rAcc := AxisCmd_rAccZ, rDec := AxisCmd_rDecZ,
    xLimEn := TRUE, rLimPos := Cfg_rLimZPos, rLimNeg := Cfg_rLimZNeg);

(* ===== R：回零 > 保持角(绝对) > 点动；M5 门控；硬限位 [Cfg_rLimRNeg, Cfg_rLimRPos] ===== *)
fbR(Axis := Axis_4, xEnable := AxisCmd_xPower AND xM5Ready, xStop := AxisCmd_xStopAll, xResetFault := AxisCmd_xResetFault,
    xHome := AxisCmd_xHomeR,
    xMoveAbs := AxisCmd_xHoldR, rTargetPos := AxisCmd_rRHoldPos,
    xJogPos := AxisCmd_xJogRPos, xJogNeg := AxisCmd_xJogRNeg, rJogVel := AxisCmd_rJogVelR,
    rVel := AxisCmd_rJogVelR, rAcc := AxisCmd_rAccR, rDec := AxisCmd_rDecR,
    xLimEn := TRUE, rLimPos := Cfg_rLimRPos, rLimNeg := Cfg_rLimRNeg);

(* ===== Y/Z/R 反馈回写 ===== *)
AxisFb_rPosY := fbY.rActPos; AxisFb_rPosZ := fbZ.rActPos; AxisFb_rPosR := fbR.rActPos;
AxisFb_xMovingY := fbY.xMoving; AxisFb_xMovingZ := fbZ.xMoving; AxisFb_xMovingR := fbR.xMoving;
AxisFb_xStandstillY := fbY.xStandstill; AxisFb_xStandstillZ := fbZ.xStandstill; AxisFb_xStandstillR := fbR.xStandstill;
AxisFb_xPoweredY := fbY.xPowered; AxisFb_xPoweredZ := fbZ.xPowered; AxisFb_xPoweredR := fbR.xPowered;
AxisFb_xReadyY := fbY.xReady; AxisFb_xReadyZ := fbZ.xReady; AxisFb_xReadyR := fbR.xReady;
AxisFb_xHomedY := fbY.xHomed; AxisFb_xHomedZ := fbZ.xHomed; AxisFb_xHomedR := fbR.xHomed;
AxisFb_xFaultY := fbY.xFault; AxisFb_xFaultZ := fbZ.xFault; AxisFb_xFaultR := fbR.xFault;
AxisFb_xReady := AxisFb_xReadyM1 AND AxisFb_xReadyM2 AND fbY.xReady AND fbZ.xReady
    AND (NOT xM5Ready OR fbR.xReady);
          
END_PROGRAM

FUNCTION_BLOCK FB_XDual
  VAR_INPUT
    xEnable : BOOL;
    xStop : BOOL;
    xResetFault : BOOL;
    xJogPos : BOOL;
    xJogNeg : BOOL;
    xSpinLeft : BOOL;
    xSpinRight : BOOL;
    xMoveRel : BOOL;
    rMoveDist : REAL;
    rMoveVel : REAL;
    rJogVel : REAL;
    rSpinVel : REAL;
    rHeadingErr : REAL;
    rKpTrack : REAL;
    rAcc : REAL;
    rDec : REAL;
    rTrimMax : REAL;
    xSyncEnable : BOOL := TRUE;
  END_VAR
  VAR_OUTPUT
    xMoveDone : BOOL;
    rPosV : REAL;
    rSyncErr : REAL;
    rVelFactor : REAL;
    xCoupled : BOOL;
    xInGearM1 : BOOL;
    xInGearM2 : BOOL;
    xPoweredV : BOOL;
    xSyncWarn : BOOL;
    xSyncFault : BOOL;
    iState : INT;
    iHoldState : INT;
    eSlaveMode : INT;
    rVelCmdM1 : REAL;
    rVelCmdM2 : REAL;
    rPosM1 : REAL;
    rPosM2 : REAL;
    xMovingM1 : BOOL;
    xMovingM2 : BOOL;
    xStandstillM1 : BOOL;
    xStandstillM2 : BOOL;
    xPoweredM1 : BOOL;
    xPoweredM2 : BOOL;
    xReadyM1 : BOOL;
    xReadyM2 : BOOL;
    xFaultM1 : BOOL;
    xFaultM2 : BOOL;
    xVelReqM1 : BOOL;
    xVelReqM2 : BOOL;
    xVelBusyM1 : BOOL;
    xVelBusyM2 : BOOL;
    xErrPowerM1 : BOOL;
    xErrPowerM2 : BOOL;
    xErrVelM1 : BOOL;
    xErrVelM2 : BOOL;
  END_VAR
  VAR
    fbPowerM1 : MC_Power;
    fbPowerM2 : MC_Power;
    fbResetM1 : MC_Reset;
    fbResetM2 : MC_Reset;
    fbJogM1 : MC_Jog;
    fbVelM1 : MC_MoveVelocity;
    fbVelM2 : MC_MoveVelocity;
    fbHaltM1 : MC_Halt;
    fbHaltM2 : MC_Halt;
    fbStopM1 : MC_Stop;
    fbStopM2 : MC_Stop;
    eDirM1 : MC_DIRECTION;
    eDirM2 : MC_DIRECTION;
    eMode : INT;
    eModePrev : INT;
    rBase : REAL;
    rVelActM1 : REAL;
    rVelActM2 : REAL;
    rTrim : REAL;
    rTrimPos : REAL;
    rKpSync : REAL := 0.1;
    rSyncDeadband : REAL := 0.05;
    rTrimPosMax : REAL := 0.15;
    rTrimPosStep : REAL := 0.02;
    rTrimPosTgt : REAL;
    rTrimPosLast : REAL;
    tonStillM1 : TON;
    tonStillM2 : TON;
    tonHoldFallback : TON;
    rHoldVelMax : REAL := 0.5;
    xSoftHold : BOOL;
    xSoftHoldPrev : BOOL;
    xSoftHoldExit : BOOL;
    xSoftHoldLatched : BOOL;
    fbSetPosM1 : MC_SetPosition;
    fbSetPosM2 : MC_SetPosition;
    xZeroGate : BOOL;
    tonZeroDelay : TON;
    xZeroReady : BOOL;
    xZeroPulsePrev : BOOL;
    xSetPosReq : BOOL;
    xPosZeroed : BOOL;
    xErrSetPosM1 : BOOL;
    xErrSetPosM2 : BOOL;
    xResetEdge : BOOL;
    xResetPrev : BOOL;
    xDirFlipM2 : BOOL;
    xVelRunPrevM2 : BOOL;
    rVelInPrevM2 : REAL;
    xM1Decel : BOOL;
    xM2Decel : BOOL;
    xBothPowered : BOOL;
    xPowerGate : BOOL;
    xReqJogM1 : BOOL;
    xReqVelM1 : BOOL;
    xReqVelM2 : BOOL;
    xNeedStopM1 : BOOL;
    xNeedStopM2 : BOOL;
    xHaltM1Prev : BOOL;
    xHaltM2Prev : BOOL;
    xMovePrev : BOOL;
    xArmed : BOOL;
    rStart : REAL;
    rAvg : REAL;
    rSyncWarnLevel : REAL := 0.05;
    rSyncFaultLevel : REAL := 0.15;
    tonSyncFault : TON;
    rAccUse : REAL;
    rDecUse : REAL;
    rAccSoftMin : REAL := 0.8;
  END_VAR
  VAR_IN_OUT
    AxisM1 : AXIS_REF_SM3;
    AxisM2 : AXIS_REF_SM3;
  END_VAR

            (* ==============================================================================
 * FB_XDual — X 轴双驱（g 线 0.32）：M1 位置主轴 + M2 速度跟随
 * 铁律：X 轴（Axis/Axis_1）只允许经本 FB 驱动；FB_Servo 不得持有 X 轴实例。
 *
 * 0.32 根因：0.26–0.31 双 MoveVelocity + 对称 trim 让两侧互相改速，
 *   位置误差积分后对打 → 前进摇晃。现场 0.2x（M1 Jog/CSP + M2 CSV）直行不晃。
 *
 * 架构：
 *   - M1：Jog 用 MC_Jog（位置轨迹）；走距/旋转用 MC_MoveVelocity
 *   - M2：CSV 跟随 M1 指令速度；视觉/轻同步只改 M2
 *   - 换向：M2 符号变化撤 Execute 一拍（对齐 FB_Servo）
 *   - 松手：撤 M2 Execute → 双轴 MC_Halt
 *   - SoftHold：保持调节器；Reset 仅手动
 *   - 同步误差：线轴直接差分（无 ±180 折算）
 * 设备树建议：M1 = CSP(8)，M2 = CSV(9)
 * ============================================================================== *)

rVelFactor := 0.0;
xCoupled := FALSE;
xInGearM1 := FALSE;
xInGearM2 := FALSE;
xPoweredV := FALSE;
eSlaveMode := 0;

(* ------------------- 1. 模式 ------------------- *)
IF xStop OR NOT xEnable THEN
    eMode := 0;
    rBase := 0.0;
ELSIF xSpinLeft XOR xSpinRight THEN
    IF xSpinLeft THEN
        eMode := 2;
    ELSE
        eMode := 3;
    END_IF;
    rBase := 0.0;
ELSIF (xJogPos XOR xJogNeg) OR xMoveRel THEN
    eMode := 1;
    IF xMoveRel THEN
        IF rMoveDist >= 0.0 THEN
            rBase := ABS(rMoveVel);
        ELSE
            rBase := -ABS(rMoveVel);
        END_IF;
    ELSIF xJogPos THEN
        rBase := ABS(rJogVel);
    ELSE
        rBase := -ABS(rJogVel);
    END_IF;
ELSE
    eMode := 0;
    rBase := 0.0;
END_IF;
iState := eMode;
IF eMode <> eModePrev THEN
    rTrimPosLast := 0.0;
    rTrimPos := 0.0;
END_IF;
eModePrev := eMode;

(* ------------------- 2. 回读 + SoftHold ------------------- *)
rPosM1 := LREAL_TO_REAL(AxisM1.fActPosition);
rPosM2 := LREAL_TO_REAL(AxisM2.fActPosition);
rVelActM1 := LREAL_TO_REAL(AxisM1.fActVelocity);
rVelActM2 := LREAL_TO_REAL(AxisM2.fActVelocity);
rAvg := (rPosM1 + rPosM2) * 0.5;
rPosV := rAvg;
rSyncErr := rPosM1 - rPosM2;

xStandstillM1 := AxisM1.nAxisState = SMC_AXIS_STATE.standstill;
xStandstillM2 := AxisM2.nAxisState = SMC_AXIS_STATE.standstill;
xMovingM1 := AxisM1.fActVelocity > 0.01 OR AxisM1.fActVelocity < -0.01;
xMovingM2 := AxisM2.fActVelocity > 0.01 OR AxisM2.fActVelocity < -0.01;

tonStillM1(IN := NOT xMovingM1, PT := T#200MS);
tonStillM2(IN := NOT xMovingM2, PT := T#200MS);
tonHoldFallback(IN := (eMode = 0) AND NOT xStop AND xEnable
                    AND (ABS(rVelActM1) < rHoldVelMax) AND (ABS(rVelActM2) < rHoldVelMax),
                PT := T#2S);
IF xStop OR NOT xEnable OR (eMode <> 0) THEN
    iHoldState := 0;
    xSoftHoldLatched := FALSE;
ELSIF xSoftHoldLatched THEN
    iHoldState := 2;
ELSIF (tonStillM1.Q AND tonStillM2.Q) OR tonHoldFallback.Q THEN
    iHoldState := 2;
    xSoftHoldLatched := TRUE;
ELSE
    iHoldState := 1;
END_IF;
xSoftHoldExit := xSoftHoldPrev AND NOT (iHoldState = 2);
xSoftHold := iHoldState = 2;
xSoftHoldPrev := xSoftHold;

xSyncWarn := ABS(rSyncErr) > rSyncWarnLevel;
tonSyncFault(IN := ABS(rSyncErr) > rSyncFaultLevel, PT := T#500MS);
IF tonSyncFault.Q THEN
    xSyncFault := TRUE;
END_IF;

(* ------------------- 3. 复位（仅手动） ------------------- *)
fbResetM1(Axis := AxisM1, Execute := xResetFault);
fbResetM2(Axis := AxisM2, Execute := xResetFault);
IF xResetFault THEN
    xSyncFault := FALSE;
END_IF;

(* ------------------- 4. 使能：SoftHold 保持调节器 ------------------- *)
fbPowerM1(Axis := AxisM1, Enable := xEnable AND NOT xStop,
          bRegulatorOn := xEnable AND NOT xStop, bDriveStart := TRUE);
fbPowerM2(Axis := AxisM2, Enable := xEnable AND NOT xStop,
          bRegulatorOn := xEnable AND NOT xStop, bDriveStart := TRUE);

xPoweredM1 := fbPowerM1.Status OR xSoftHold;
xPoweredM2 := fbPowerM2.Status OR xSoftHold;
xFaultM1 := AxisM1.bError AND NOT (xSoftHold OR (iHoldState = 1));
xFaultM2 := AxisM2.bError AND NOT (xSoftHold OR (iHoldState = 1));
xReadyM1 := xPoweredM1 AND NOT xFaultM1;
xReadyM2 := xPoweredM2 AND NOT xFaultM2;
xBothPowered := xPoweredM1 AND xPoweredM2;
xPowerGate := (xEnable AND NOT xStop AND NOT xFaultM1 AND NOT xFaultM2) OR xM1Decel OR xM2Decel;

(* ------------------- 5. 置零 ------------------- *)
xZeroGate := xEnable AND xBothPowered AND NOT xPosZeroed;
tonZeroDelay(IN := xZeroGate, PT := T#500MS);
xZeroReady := tonZeroDelay.Q AND NOT xZeroPulsePrev;
xZeroPulsePrev := tonZeroDelay.Q;

xResetEdge := xResetFault AND NOT xResetPrev;
xResetPrev := xResetFault;

IF xZeroReady OR xResetEdge THEN
    xSetPosReq := TRUE;
END_IF;
fbSetPosM1(Axis := AxisM1, Execute := xSetPosReq, Position := 0.0);
fbSetPosM2(Axis := AxisM2, Execute := xSetPosReq, Position := 0.0);
xErrSetPosM1 := fbSetPosM1.Error;
xErrSetPosM2 := fbSetPosM2.Error;
IF xSetPosReq THEN
    IF (fbSetPosM1.Done AND fbSetPosM2.Done) OR fbSetPosM1.Error OR fbSetPosM2.Error THEN
        xSetPosReq := FALSE;
        xPosZeroed := TRUE;
        rTrimPosLast := 0.0;
        rTrimPos := 0.0;
    END_IF;
END_IF;

(* ------------------- 6. 指令：M1 主轴不改速，M2 跟随 ------------------- *)
CASE eMode OF
    1:
        rVelCmdM1 := rBase;
    2:
        rVelCmdM1 := ABS(rSpinVel);
    3:
        rVelCmdM1 := -ABS(rSpinVel);
ELSE
    rVelCmdM1 := 0.0;
END_CASE;

IF (eMode = 1) AND xSyncEnable THEN
    IF ABS(rSyncErr) > rSyncDeadband THEN
        rTrimPosTgt := rKpSync * rSyncErr;
    ELSE
        rTrimPosTgt := 0.0;
    END_IF;
    IF ABS(rBase) > 0.001 THEN
        IF ABS(rTrimPosTgt) > (0.4 * ABS(rBase)) THEN
            IF rTrimPosTgt > 0.0 THEN
                rTrimPosTgt := 0.4 * ABS(rBase);
            ELSE
                rTrimPosTgt := -0.4 * ABS(rBase);
            END_IF;
        END_IF;
    END_IF;
    rTrimPosTgt := LIMIT(-ABS(rTrimPosMax), rTrimPosTgt, ABS(rTrimPosMax));
    rTrimPos := LIMIT(rTrimPosLast - rTrimPosStep, rTrimPosTgt, rTrimPosLast + rTrimPosStep);
    rTrimPosLast := rTrimPos;
ELSE
    rTrimPos := 0.0;
    rTrimPosLast := 0.0;
END_IF;

IF eMode = 1 THEN
    rTrim := LIMIT(-ABS(rTrimMax), rKpTrack * rHeadingErr, ABS(rTrimMax));
    rVelCmdM2 := rVelCmdM1 - 2.0 * rTrim + rTrimPos;
    IF ABS(rVelCmdM1) > 0.001 THEN
        IF rVelCmdM1 > 0.0 THEN
            IF rVelCmdM2 < 0.0 THEN
                rVelCmdM2 := 0.0;
            END_IF;
        ELSE
            IF rVelCmdM2 > 0.0 THEN
                rVelCmdM2 := 0.0;
            END_IF;
        END_IF;
    END_IF;
ELSIF (eMode = 2) OR (eMode = 3) THEN
    rTrim := 0.0;
    rVelCmdM2 := -rVelCmdM1;
ELSE
    rTrim := 0.0;
    rVelCmdM2 := 0.0;
END_IF;
IF xStop OR NOT xEnable THEN
    rVelCmdM1 := 0.0;
    rVelCmdM2 := 0.0;
    rTrimPosLast := 0.0;
    rTrimPos := 0.0;
END_IF;

rAccUse := ABS(rAcc);
IF rAccUse < rAccSoftMin THEN
    rAccUse := rAccSoftMin;
END_IF;
rDecUse := ABS(rDec);
IF rDecUse < rAccSoftMin THEN
    rDecUse := rAccSoftMin;
END_IF;

(* ------------------- 7. M1：Jog / MoveVelocity ------------------- *)
xReqJogM1 := (eMode = 1) AND NOT xMoveRel AND xPowerGate AND NOT xSoftHold
             AND (ABS(rJogVel) > 0.001);
xReqVelM1 := (((eMode = 1) AND xMoveRel) OR (eMode = 2) OR (eMode = 3))
             AND xPowerGate AND NOT xSoftHold AND (ABS(rVelCmdM1) > 0.001);

IF rVelCmdM1 >= 0.0 THEN
    eDirM1 := positive;
ELSE
    eDirM1 := negative;
END_IF;

fbJogM1(Axis := AxisM1,
        JogForward := xReqJogM1 AND xJogPos,
        JogBackward := xReqJogM1 AND xJogNeg,
        Velocity := ABS(rJogVel), Acceleration := rAccUse, Deceleration := rDecUse);
fbVelM1(Axis := AxisM1, Execute := xReqVelM1,
        Velocity := ABS(rVelCmdM1), Direction := eDirM1,
        Acceleration := rAccUse, Deceleration := rDecUse);

(* ------------------- 8. M2：速度跟随（松手立刻撤 Execute） ------------------- *)
IF (eMode = 0) OR (NOT xPowerGate) OR xSoftHold OR xStop OR (ABS(rVelCmdM2) <= 0.001) THEN
    xReqVelM2 := FALSE;
ELSE
    xReqVelM2 := TRUE;
END_IF;

xM1Decel := (NOT xReqJogM1) AND (NOT xReqVelM1) AND xPowerGate
            AND xMovingM1 AND NOT xStop AND NOT xSoftHold;
xM2Decel := (NOT xReqVelM2) AND xPowerGate AND xMovingM2 AND NOT xStop AND NOT xSoftHold;

IF rVelCmdM2 >= 0.0 THEN
    eDirM2 := positive;
ELSE
    eDirM2 := negative;
END_IF;

xDirFlipM2 := xReqVelM2 AND xVelRunPrevM2 AND ((rVelCmdM2 >= 0.0) <> (rVelInPrevM2 >= 0.0));
fbVelM2(Axis := AxisM2, Execute := xReqVelM2 AND NOT xDirFlipM2,
        Velocity := ABS(rVelCmdM2), Direction := eDirM2,
        Acceleration := rAccUse, Deceleration := rDecUse);
xVelRunPrevM2 := xReqVelM2;
rVelInPrevM2 := rVelCmdM2;

(* ------------------- 9. 停车 ------------------- *)
fbStopM1(Axis := AxisM1, Execute := xStop, Deceleration := rDecUse);
fbStopM2(Axis := AxisM2, Execute := xStop, Deceleration := rDecUse);

xNeedStopM1 := xPowerGate AND NOT xSoftHold AND NOT xStop AND NOT xReqJogM1 AND NOT xReqVelM1;
xNeedStopM2 := xPowerGate AND NOT xSoftHold AND NOT xStop AND NOT xReqVelM2;
fbHaltM1(Axis := AxisM1, Execute := xNeedStopM1 AND xMovingM1 AND NOT xHaltM1Prev,
         Deceleration := rDecUse);
fbHaltM2(Axis := AxisM2, Execute := xNeedStopM2 AND xMovingM2 AND NOT xHaltM2Prev,
         Deceleration := rDecUse);
xHaltM1Prev := xNeedStopM1 AND (xMovingM1 OR NOT tonStillM1.Q);
xHaltM2Prev := xNeedStopM2 AND (xMovingM2 OR NOT tonStillM2.Q);

(* ------------------- 10. 诊断与走距完成 ------------------- *)
xVelReqM1 := xReqVelM1;
xVelReqM2 := xReqVelM2;
xVelBusyM1 := fbVelM1.Busy;
xVelBusyM2 := fbVelM2.Busy;
xErrPowerM1 := fbPowerM1.Error;
xErrPowerM2 := fbPowerM2.Error;
xErrVelM1 := fbVelM1.Error;
xErrVelM2 := fbVelM2.Error;

IF xStop OR NOT xEnable OR NOT xMoveRel THEN
    xArmed := FALSE;
    xMoveDone := FALSE;
ELSE
    IF xMoveRel AND NOT xMovePrev THEN
        xArmed := TRUE;
        rStart := rAvg;
    END_IF;
    xMoveDone := xArmed AND (ABS(rAvg - rStart) >= ABS(rMoveDist));
END_IF;
xMovePrev := xMoveRel;
          
END_FUNCTION_BLOCK

CONFIGURATION Device
END_CONFIGURATION

CONFIGURATION HIGH_SPEED_IO
END_CONFIGURATION

CONFIGURATION ETHERCAT
END_CONFIGURATION

CONFIGURATION MDX_EC
END_CONFIGURATION

CONFIGURATION Axis
END_CONFIGURATION

CONFIGURATION MDX_EC_1
END_CONFIGURATION

CONFIGURATION Axis_1
END_CONFIGURATION

CONFIGURATION MDX_EC_2
END_CONFIGURATION

CONFIGURATION Axis_2
END_CONFIGURATION

CONFIGURATION MDX_EC_3
END_CONFIGURATION

CONFIGURATION Axis_3
END_CONFIGURATION

CONFIGURATION MDX_EC_4
END_CONFIGURATION

CONFIGURATION Axis_4
END_CONFIGURATION

CONFIGURATION MODBUS_COM0
END_CONFIGURATION

CONFIGURATION modbus_protocol
END_CONFIGURATION

CONFIGURATION MODBUS_TCP
END_CONFIGURATION
